// ---- Hardware/NanotecPanDrive/FB_NanotecPD_Home.TcPOU
FUNCTION_BLOCK FB_NanotecPD_Home
VAR_INPUT
	bExecute 	: BOOL;
	bStop		: BOOL;
END_VAR
VAR_OUTPUT
	bBusy 		: BOOL;
	bError 		: BOOL;
	nErrorId 	: ERRORID;	
END_VAR
VAR_IN_OUT
	pHwRef : POINTER TO FB_HwRefNanotecPD; 
END_VAR
VAR
	nState 				: USINT;
	nStateNext			: USINT;
	fbSdoWrite 			: FB_SDO_WRITE;
	eCurrentHomingState : E_CoDS402HomingState;
END_VAR

IF bExecute THEN
	CASE nState OF
		0:	//Set fast homing speed
			bBusy := TRUE;
			fbSdoWrite.nIndex := 16#6099;
			fbSdoWrite.nSubIndex := 1;
			fbSdoWrite.nDataLength := 4;
			fbSdoWrite.nData := pHwRef^.M_RealToInternSpeed(pHwRef^.P_nFastHomingSpeed);
			nState := 40;
			nStateNext := 1;
			
		1:	//Set slow homing speed
			fbSdoWrite.nIndex := 16#6099;
			fbSdoWrite.nSubIndex := 2;
			fbSdoWrite.nDataLength := 4;
			fbSdoWrite.nData := pHwRef^.M_RealToInternSpeed(pHwRef^.P_nSlowHomingSpeed);
			nState := 40;
			nStateNext := 2;
			
		2:	//Set homing methode
			fbSdoWrite.nIndex := 16#6098;
			fbSdoWrite.nSubIndex := 0;
			fbSdoWrite.nDataLength := 1;
			IF pHwRef^.P_bInvertInitDir THEN
				fbSdoWrite.nData := 2;
			ELSE
				fbSdoWrite.nData := 1;
			END_IF
			nState := 40;
			nStateNext := 3;
			
		3: 	//Write home offset
			fbSdoWrite.nIndex := 16#607C;
			fbSdoWrite.nSubIndex := 0;
			fbSdoWrite.nDataLength := 4;
			//Hier braucht es Umrechnung von Real to intern Pos
			fbSdoWrite.nData := pHwRef^.M_RealToInternPos(pHwRef^.P_nRefPos);
			nState := 40;
			IF pHwRef^.M_GetDS402State() = E_CoDS402States.DS402STATE_OperationEnabled THEN
				nStateNext := 4;
			ELSE
				nStateNext := 5;
			END_IF
			
		4:	//Mode lässt sich nicht in "OperationEnabled" setzen
			pHwRef^.nControlword := 7;
			IF pHwRef^.M_GetDS402State() = E_CoDS402States.DS402STATE_SwitchedOn THEN
				nState := 5;	
			END_IF
			
		5:	//Set Mode of operation to "6" (Homing)
			pHwRef^.nMode := 6; //Homing
			IF pHwRef^.nCurrentMode = 6 THEN
				nState := 6;	
			END_IF

		6:	//Statemachine in "OperationEnabled" setzen
			pHwRef^.nControlword := 15;
			IF pHwRef^.M_GetDS402State() = E_CoDS402States.DS402STATE_OperationEnabled THEN
				nState := 7;
			END_IF
			
		7:	//Start homing
			pHwRef^.nControlword := 31;
			eCurrentHomingState := pHwRef^.M_GetHomingState();
			IF eCurrentHomingState = E_CoDS402HomingState.HomingInProgress THEN
				nState := 8;
			END_IF
			
		8:	//Wait for State "Homing in process
			IF pHwRef^.M_GetDS402State() = E_CoDS402States.DS402STATE_OperationEnabled THEN
				IF bStop THEN
					pHwRef^.nControlword := 15;
					nState := 80;
				ELSE
					eCurrentHomingState := pHwRef^.M_GetHomingState();
					CASE eCurrentHomingState OF
						E_CoDS402HomingState.HomingAttainedButNotReached,
						E_CoDS402HomingState.HomingError,
						E_CoDS402HomingState.HomingInteruptedOrNotReached:
							nErrorId := E_ErrorIdDS402.ERRORID_HomingInterruptedOrNotReached;
							nState := 99;
						E_CoDS402HomingState.HomingSuccess:
							pHwRef^.P_bIsHomed := TRUE;
							pHwRef^.nControlword := 7;
							pHwRef^.nMode := 1;
							pHwRef^.nTargetSpeed := DINT_TO_INT(pHwRef^.M_RealToInternSpeed(pHwRef^.P_nFastHomingSpeed));
							pHwRef^.nTargetPosition := pHwRef^.M_RealToInternPos(pHwRef^.P_nHomePos);
							nState := 9;
					END_CASE
				END_IF
			ELSE
				nErrorId := E_ErrorIdDS402.ERRORID_OperationNotEnabled;
				nState := 99;
			END_IF
			
		9:	//Move to WorkingPos1
			IF pHwRef^.nCurrentMode = 1 THEN
				pHwRef^.nControlword := 15;
				nState := 10;
			END_IF
			
		10:	IF pHwRef^.M_GetDS402State() = E_CoDS402States.DS402STATE_OperationEnabled THEN
				pHwRef^.nControlword := 31;
				nState := 11;
			END_IF
			
		11:	//Wait for setpoint acknowledge
			IF pHwRef^.nStatusword.12 THEN
				pHwRef^.nControlword := 15;
				nState := 12;
			END_IF
			
		12:	//Wait for target reached
			IF pHwRef^.M_GetDS402State() = E_CoDS402States.DS402STATE_OperationEnabled THEN
				IF bStop THEN
					pHwRef^.nControlword.8 := TRUE;
					nState := 13;
				ELSE
					IF pHwRef^.nStatusword.10 THEN
						nState := 80;	
					END_IF
				END_IF
			ELSE
				nErrorId := E_ErrorIdDS402.ERRORID_OperationNotEnabled;
				nState := 99;
			END_IF
			
		13:	//Warten bis Motor sich nicht mehr dreht -> dann Power-STM in SwitchedOn setzen, damit Fahrauftrag gelöscht wird
			IF pHwRef^.nCurrentSpeed = 0 THEN
				pHwRef^.nControlword := 7;
				nState := 14;
			END_IF
			
		14:	//Power-STM wieder in OperationEnable setzen
			IF pHwRef^.M_GetDS402State() = E_CoDS402States.DS402STATE_SwitchedOn THEN
				pHwRef^.nControlword := 15;
				pHwRef^.P_bIsHomed := TRUE;
				nState := 80;
			END_IF		

	END_CASE
	
	//Sdo senden
	IF nState = 40 THEN
		fbSdoWrite(sADSNetID:= pHwRef^.P_sAdsNetId, nPortNr:= pHwRef^.P_nAdsPort, bExecute:= TRUE);
		IF NOT fbSdoWrite.bBusy THEN
			IF fbSdoWrite.bError THEN
				nErrorId := fbSdoWrite.nAdsErrorId;
				nState := 99;
			ELSE
				nState := nStateNext;
			END_IF
			fbSdoWrite(bExecute:= FALSE);
		END_IF		
	END_IF
	
	IF nState >= 80 THEN
		bBusy := FALSE;
		IF nState = 99 THEN
			bError := TRUE;
		END_IF
	END_IF
	
ELSE
	bError := FALSE;
	nErrorId := 0;
	nState := 0;	
END_IF

END_FUNCTION_BLOCK

// ---- Hardware/TMCM-1140/FB_TMCM1140_Home.TcPOU
FUNCTION_BLOCK FB_TMCM1140_Home
VAR_INPUT
	bExecute	: BOOL;
	bStop		: BOOL;
END_VAR
VAR_OUTPUT
	bBusy 		: BOOL;
	bError 		: BOOL;
	nErrorId 	: ERRORID;	
END_VAR
VAR_IN_OUT
	pHwRef : POINTER TO FB_HwRefTMCM1140;
END_VAR
VAR
	nState 			: USINT;
	nStateNext 		: USINT;
	bDigiout0 		: BOOL;
	bDigiout1 		: BOOL;
	fbSdoWrite 		: FB_SDO_WRITE;
	eCurrentHomingState : E_CoDS402HomingState;
END_VAR

IF bExecute THEN
	CASE nState OF
		0:	//Set Fast homing speed
			bBusy := TRUE;
			fbSdoWrite.nIndex := 16#6099;
			fbSdoWrite.nSubIndex := 1;
			fbSdoWrite.nDataLength := 4;
			fbSdoWrite.nData := pHwRef^.M_RealToInternSpeed(pHwRef^.P_nFastHomingSpeed);
			nState := 40;
			nStateNext := 1;
			
		1:	//Set Slow homing speed
			fbSdoWrite.nIndex := 16#6099;
			fbSdoWrite.nSubIndex := 2;
			fbSdoWrite.nDataLength := 4;
			fbSdoWrite.nData := pHwRef^.M_RealToInternSpeed(pHwRef^.P_nSlowHomingSpeed);
			nState := 40;
			nStateNext := 2;			

		2:	//Set homing methode
			fbSdoWrite.nIndex := 16#6098;
			fbSdoWrite.nSubIndex := 0;
			fbSdoWrite.nDataLength := 1;
			fbSdoWrite.nData := pHwRef^.P_eHomingMethode;
			nState := 40;
			nStateNext := 3;
			
		3: 	//Write home offset
			fbSdoWrite.nIndex := 16#607C;
			fbSdoWrite.nSubIndex := 0;
			fbSdoWrite.nDataLength := 4;
			fbSdoWrite.nData := pHwRef^.M_RealToInternPos(pHwRef^.P_nRefPos);
			nState := 40;
			nStateNext := 4;
			
		4:	//Write profile speed
			fbSdoWrite.nIndex := 16#6081;
			fbSdoWrite.nSubIndex := 0;
			fbSdoWrite.nDataLength := 4;
			fbSdoWrite.nData := pHwRef^.M_RealToInternSpeed(pHwRef^.P_nMaxSpeed);
			nState := 40;
			nStateNext := 5;

		5:	//Set Mode of operation to "6" (Homing)
			pHwRef^.nMode := 6; //Homing
			nState := 6;
			
		6:	//Start homing
			pHwRef^.nControlword := 31;
			nState := 7;
			
		7:	//Wait for State "Homing in process
			IF pHwRef^.M_GetDS402State() = E_CoDS402States.DS402STATE_OperationEnabled THEN
				IF bStop THEN
					pHwRef^.nControlword := 15;
					nState := 80;
				ELSE
					eCurrentHomingState := pHwRef^.M_GetHomingState();
					CASE eCurrentHomingState OF
						E_CoDS402HomingState.HomingAttainedButNotReached,
						E_CoDS402HomingState.HomingError,
						E_CoDS402HomingState.HomingInteruptedOrNotReached:
							nErrorId := E_ErrorIdDS402.ERRORID_HomingInterruptedOrNotReached;
							nState := 99;
						E_CoDS402HomingState.HomingSuccess:
							pHwRef^.nControlword := 15;
							pHwRef^.nMode := 1;	//PP mode
							pHwRef^.M_SetTargetPos(pHwRef^.P_nHomePos, FALSE);
							pHwRef^.P_bIsHomed := TRUE;
							nState := 8;
					END_CASE
				END_IF
			ELSE
				nErrorId := 43434;
				nState := 99;
			END_IF
			
		8:	//Move to HomePos
			pHwRef^.nControlword := 31;
			nState := 9;
			
		9:	//Wait for setpoint acknowledge
			IF pHwRef^.nStatusword.12 THEN
				pHwRef^.nControlword := 15;
				nState := 10;
			END_IF
			
		10:	//Wait for target reached
			IF pHwRef^.M_GetDS402State() = E_CoDS402States.DS402STATE_OperationEnabled THEN
				//Das HALT-Bit von von der TMCM1140 nicht unterstützt.
				//Man kann den Mode auf "0" setzen und dann sollter der Motor auch anhalten
				IF bStop THEN
					IF bStop THEN
						pHwRef^.nMode := 0;
						nState := 80;
					END_IF
				ELSE
					IF pHwRef^.nStatusword.10 THEN
						nState := 80;
					END_IF
				END_IF
			ELSE
				nErrorId := E_ErrorIdDS402.ERRORID_OperationNotEnabled;
				nState := 99;
			END_IF
			
	END_CASE
	
	//Sdo senden
	IF nState = 40 THEN
		fbSdoWrite(sADSNetID:= pHwRef^.P_sAdsNetId, nPortNr:= pHwRef^.P_nAdsPort, bExecute:= TRUE);
		IF NOT fbSdoWrite.bBusy THEN
			IF fbSdoWrite.bError THEN
				nErrorId := fbSdoWrite.nAdsErrorId;
				nState := 99;
			ELSE
				nState := nStateNext;
			END_IF
			fbSdoWrite(bExecute:= FALSE);
		END_IF		
	END_IF
	
	IF nState >= 80 THEN
		bBusy := FALSE;
		IF nState = 99 THEN
			bError := TRUE;
		END_IF
	END_IF

ELSE
	bBusy 	:= FALSE;
	bError 	:= FALSE;
	bStop 	:= FALSE;
	nState 	:= 0;
END_IF

END_FUNCTION_BLOCK

// ---- Hardware/NanotecPanDrive/FB_NanotecPD_Move.TcPOU
FUNCTION_BLOCK FB_NanotecPD_Move
VAR_INPUT
	bExecute 	: BOOL;
	bStop		: BOOL;
	nPosition	: DINT; //Reale Einheit (µm oder 1/10°)
	nSpeed		: DINT; //Reale Einheit/s	
END_VAR
VAR_OUTPUT
	bBusy 		: BOOL;
	bError 		: BOOL;
	nErrorId 	: ERRORID;	
END_VAR
VAR_IN_OUT
	pHwRef : POINTER TO FB_HwRefNanotecPD; 
END_VAR
VAR
	nState 					: USINT;
	eCurrentCoDS402State 	: E_CoDS402States;
	fbGetCurrTaskIndex		: GETCURTASKINDEX;
	nCurrentTaskCycleCount 	: UDINT;	
END_VAR

IF bExecute THEN
	eCurrentCoDS402State := pHwRef^.M_GetDS402State();
	
	CASE nState OF
		0:	//Vorbedingungen prüfen
			bBusy := TRUE;
			nState := 1;
			IF pHwRef^.bError THEN
				nErrorID := E_ErrorIdHwGeneral.ERRORID_DriveIsInErrorState;
				nState := 99;
			ELSE
				IF pHwRef^.bBusy THEN
					nErrorID := E_ErrorIdHwGeneral.ERRORID_DriveIsStillBusy;
					nState := 99;
				ELSE
					IF NOT pHwRef^.P_bIsHomed THEN
						nErrorID := E_ErrorIdHwGeneral.ERRORID_DriveNotHomed;
						nState := 99;
					ELSE
						IF NOT pHwRef^.M_SetTargetPos(nPosition) THEN
							nErrorID := E_ErrorIdHwGeneral.ERRORID_InvalidPosition;
							nState := 99;
						ELSE
							IF NOT pHwRef^.M_SetTargetSpeed(nSpeed) THEN
								nErrorID := E_ErrorIdHwGeneral.ERRORID_InvalidSpeed;
								nState := 99;
							END_IF
						END_IF	
					END_IF
				END_IF
			END_IF
			
			fbGetCurrTaskIndex();
			nCurrentTaskCycleCount := TwinCAT_SystemInfoVarList._TaskInfo[fbGetCurrTaskIndex.index].CycleCount;

		1:	//Mode sollte durch Homing bereits auf 1 stehen
			//Dieser State darf niemals im gleichen Zyklus wie State 0 ausgeführt werden. Passiert wenn FB im selben Zyklus auf-
			//gerufen wird. Somit wird sichergestellt, dass die Zielposition auch im Drive eher ankommt, wie das Startbit.
			IF TwinCAT_SystemInfoVarList._TaskInfo[fbGetCurrTaskIndex.index].CycleCount <> nCurrentTaskCycleCount THEN
				IF eCurrentCoDS402State = E_CoDS402States.DS402STATE_OperationEnabled THEN
					pHwRef^.nControlword := 31;
					nState := 2;
				ELSE
					nErrorID := E_ErrorIdDS402.ERRORID_OperationNotEnabled;
					nState := 99;
				END_IF
			END_IF
			
		2:	//Setpoint ACK?
			IF pHwRef^.nStatusword.12 THEN
				pHwRef^.nControlword := 15;
				nState := 3;
			END_IF
			
		3:	//Target reached?
			IF pHwRef^.bError THEN
				nErrorId := pHwRef^.P_nErrorID;
				nState := 99;
			ELSE
				{warning 'Safety sollte noch mit abgefragt werden'}
				IF bStop THEN
					pHwRef^.nControlword.8 := TRUE;
					nState := 4;
				END_IF
				
				IF pHwRef^.nStatusword.10 THEN
					nState := 80; //Ready
				END_IF
			END_IF
			
		4:	//Warten bis Motor sich nicht mehr dreht -> dann OperationEnable zurück nehmen
			IF pHwRef^.nCurrentSpeed = 0 THEN
				pHwRef^.nControlword := 7;
				nState := 5;
			END_IF			
			
		5:	//STM wieder in OperationEnable
			IF pHwRef^.M_GetDS402State() = E_CoDS402States.DS402STATE_SwitchedOn THEN
				pHwRef^.nControlword := 15;
				nState := 80; //Ready
			END_IF
	END_CASE
	
	IF nState >= 80 THEN
		bBusy := FALSE;
		IF nState = 99 THEN
			bError := TRUE;
		END_IF
	END_IF
	
ELSE
	bError := FALSE;
	nErrorId := 0;
	nState := 0;
END_IF

END_FUNCTION_BLOCK

// ---- Hardware/TrayLock/FB_HwTrayLockControl.TcPOU
FUNCTION_BLOCK FB_HwTrayLockControl
VAR_INPUT
	bExecute		: BOOL;
	eCtrl			: E_LockCtrl;
END_VAR
VAR_OUTPUT
	bBusy 		: BOOL;
	bError 		: BOOL;
	nErrorId	: ERRORID;	
END_VAR
VAR_IN_OUT
	pHwRef : POINTER TO FB_HwRefTrayLock;
END_VAR
VAR
	nState		: USINT;
	timer		: TON;
END_VAR

IF bExecute THEN
	IF pHwRef = 0 THEN
		bError := TRUE;
		nErrorId := E_ErrorIdHwGeneral.ERRORID_InvalidHwRef;
		RETURN;
	END_IF

	CASE nState OF
		0:	IF eCtrl = E_LockCtrl.Unlock THEN
				IF pHwRef^.eCurrentState = E_LockState.Unlocked THEN
					RETURN;
				ELSE
					bBusy := TRUE;
					nState := 1; //Unlocking
				END_IF
			ELSE
				IF pHwRef^.eCurrentState = E_LockState.Locked THEN
					RETURN;
				ELSE
					bBusy := TRUE;
					nState := 10; //Locking
				END_IF
			END_IF
			
		1:	//Unlocking, disable heater
			pHwRef^.bDisableHeater := TRUE;
			timer(IN:= TRUE, PT:= T#200MS);
			nState := 2;
			
		2:	//Time elapsed?
			timer();
			IF timer.Q THEN
				timer(IN:= FALSE);
				nState := 3;
			END_IF
			
		3:	//Set outputs
			pHwRef^.bLock := FALSE;
			pHwRef^.bUnlock := TRUE;
			timer(IN:= TRUE, PT:= T#3S); //Timeout
			IF pHwRef^.P_bFeedback THEN
				IF pHwRef^.bUnlocked THEN
					nState := 80;
				ELSIF timer.Q THEN
					nErrorId := E_ErrorIdHwGeneral.ERRORID_UnlockingFailed;
					nState := 99; //Error
				END_IF
			ELSE
				IF timer.Q THEN
					nState := 80;
				END_IF
			END_IF
			
		10: //Locking
			pHwRef^.bLock := TRUE;
			pHwRef^.bUnlock := FALSE;
			timer(IN:= TRUE, PT:= T#3S); //Timeout
			IF pHwRef^.P_bFeedback THEN
				IF pHwRef^.bLocked THEN
					//Enable heater
					pHwRef^.bDisableHeater := FALSE;
					nState := 80;
				ELSIF timer.Q THEN
					nErrorId := E_ErrorIdHwGeneral.ERRORID_LockingFailed;
					nState := 99; //Error
				END_IF
			ELSE
				IF timer.Q THEN
					nState := 80;
				END_IF
			END_IF
	END_CASE
	
	IF nState >= 80 THEN
		pHwRef^.bLock := FALSE;
		pHwRef^.bUnlock := FALSE;
		bBusy := FALSE;
		IF nState = 99 THEN
			bError := TRUE;
		END_IF
	END_IF

ELSE
	timer(IN:= FALSE);
	bBusy := FALSE;
	bError := FALSE;
	nErrorId := 0;
	nState := 0;	
END_IF

END_FUNCTION_BLOCK

// ---- Objects/Devices/FB_Stacker.TcPOU
FUNCTION_BLOCK FB_Stacker EXTENDS FB_Object IMPLEMENTS I_Device

VAR
	nParentSlotNr		: UINT;		//Stacker befindet sich zwar an keinem Slot, aber virtuell in der GUI (am Root)#
	eCurrentState		: E_MachineState := E_MachineState.MACHINESTATE_Idle;
	nNotifyId			: UINT;
	nErrorId			: ERRORID;
	bCanceled			: BOOL;
	bStopAllOnError		: BOOL;
	bIsInit				: BOOL;
	bBusy				: BOOL;
	bError				: BOOL;
	stError				: ST_Error :=(POU := E_POU.POU_FB_Stacker);
	
	nNumberOfShelves	: USINT;
	aShelfes			: ARRAY[1..cMaxShelfes] OF ST_Shelf;
	
	//Hardware-Referenzen
	pHwRef_SpinDrive	: POINTER TO FB_HwRefEL70xxDrive;
	pHwRef_LiftDrive	: POINTER TO FB_HwRefEL70xxDrive;
	pHwRef_TrayStop		: POINTER TO FB_HwRefEL70xxDrive;
	
	bSensorTransAreaLeft 		AT %I* : BOOL;
	bSensorTransAreaRight		AT %I* : BOOL;
	bSensorTrayAlignmentLeft 	AT %I* : BOOL;
	bSensorTrayAlignmentRight 	AT %I* : BOOL;
	bSensorTrayDetection		AT %I* : BOOL;
	
	//Spec-Properties
	nLoadingPosAngle		: DINT;	//Drehwinkel Beladeposition
	nTransferPosAnglePrint1 : DINT;	//Drehwinkel Transferpostion zu Drucker 1
	nTransferPosAnglePrint2 : DINT;	//Drehwinkel Transferpostion zu Drucker 2 (wird derzeit nicht verwendet)
		
	//****************************************Aktionvariablen****************************************************
	
	//Action: "Init"
	bInit				: BOOL;
	nStateA_Init		: USINT;
	fbPower 			: FB_HWECtrl_EL70xx_Power;
	fbHoming 			: FB_HWECtrl_EL70xx_Home;
	pCurrentInitDrive	: POINTER TO FB_HwRefEL70xxDrive;
	
	//Action: "TurnTo"
	bTurnTo				: BOOL;
	nStateA_TurnTo		: USINT;
	fbHwCtrl_Turn		: FB_HWECtrl_EL70xx_Move;
	nTurnToPosition		: DINT;
	
	//Action: "MoveLifter"
	bMoveLifter			: BOOL;
	nStateA_MoveLifter	: USINT;
	nMoveLifterPosition	: DINT;
	nMoveLifterSpeed	: DINT;
	fbHWECtrl_MoveLifter: FB_HWECtrl_EL70xx_Move;
	
	//Action: "OpenCloseTrayStop"
	bOpClTrayStop			: BOOL;
	nStateA_OpClTrayStop	: USINT;
	eOpClTrayStopCtrl		: E_OpClCtrl;
	fbHwCtrl_MoveTrayStop 	: FB_HWECtrl_EL70xx_Move;
	
	//Action: "Load" (Bestücken oder Entnehmen)
	bLoad			: BOOL;
	nStateA_Load	: USINT;
	nBottomShelf	: UINT; //unterstes Fach
	
	stProcessData		: ST_ObjectProcData;
	
END_VAR

VAR CONSTANT
	cMaxShelfes : UINT := 10;
END_VAR

CASE eCurrentState OF
	E_MachineState.MACHINESTATE_Active:
	
		IF bInit THEN
			A_Init();
			IF nStateA_Init >= 80 THEN
				IF nStateA_Init >= 99 THEN
					bError := TRUE;	
				END_IF
				bInit := FALSE;
				nStateA_Init := 0;
			END_IF
		END_IF
		
		IF bTurnTo THEN
			A_TurnTo();
			IF nStateA_TurnTo >= 80 THEN
				IF nStateA_TurnTo >= 99 THEN
					bError := TRUE;	
				END_IF
				bTurnTo := FALSE;
				nStateA_TurnTo := 0;
			END_IF
		END_IF
		
		IF bMoveLifter THEN
			A_MoveLifter();
			IF nStateA_MoveLifter >= 80 THEN
				IF nStateA_MoveLifter >= 99 THEN
					bError := TRUE;	
				END_IF
				bMoveLifter := FALSE;
				nStateA_MoveLifter := 0;
			END_IF
		END_IF
		
		IF bOpClTrayStop THEN
			A_OpClTrayStop();
			IF nStateA_OpClTrayStop >= 80 THEN
				IF nStateA_OpClTrayStop >= 99 THEN
					bError := TRUE;	
				END_IF
				bOpClTrayStop := FALSE;
				nStateA_OpClTrayStop := 0;
			END_IF
		END_IF
		
		IF bLoad THEN
			A_Load();
			IF nStateA_Load >= 80 THEN
				IF nStateA_Load >= 99 THEN
					bError := TRUE;	
				END_IF
				bLoad := FALSE;
				nStateA_Load := 0;
			END_IF
		END_IF
		
		IF NOT (bInit OR bTurnTo OR bMoveLifter OR bOpClTrayStop OR bLoad) THEN
			bBusy := FALSE;
			eCurrentState := E_MachineState.MACHINESTATE_Idle;
		END_IF

		IF bError  THEN
			eCurrentState := E_MachineState.MACHINESTATE_Error;
		END_IF

	E_MachineState.MACHINESTATE_Reset:
		nStateA_Init := 0;
		nStateA_TurnTo := 0;
		nStateA_MoveLifter := 0;
		nStateA_OpClTrayStop := 0;
		nStateA_Load := 0;
		bBusy := FALSE;
		bError := FALSE;
		bStopAllOnError := FALSE;
		stError.Cmd := 0;
		stError.ErrorId := 0;
		eCurrentState := E_MachineState.MACHINESTATE_Idle;
	
	E_MachineState.MACHINESTATE_Error:
		bBusy := FALSE;
END_CASE

//Prozessdaten aktualisieren
stProcessData.nObjId := nObjectID;
stProcessData.n32Data[0] := BOOL_TO_DINT(P_bIsInit);
stProcessData.n32Data[1] := eCurrentState;
stProcessData.n32Data[2] := stError.ErrorId;
stProcessData.n32Data[3] := pHwRef_LiftDrive^.P_nActualPosition;
stProcessData.n32Data[4] := pHwRef_SpinDrive^.P_nActualPosition;
IF pHwRef_TrayStop^.bInput1 THEN //Open
	stProcessData.n32Data[5] := E_OpClState.Open;
ELSIF pHwRef_TrayStop^.bInput2 THEN //Closed
	stProcessData.n32Data[5] := E_OpClState.Closed;
ELSE
	stProcessData.n32Data[5] := E_OpClState.UNDEFINED;
END_IF
	stProcessData.n32Data[6] := BOOL_TO_DINT(bSensorTrayAlignmentLeft AND bSensorTrayAlignmentRight);

aObjProcData[nNotifyId] := stProcessData;

ACTION A_Init:
stError.POUState := nStateA_Init;

CASE nStateA_Init OF
	0:	//Power TrayStop
		pCurrentInitDrive := pHwRef_TrayStop;
		fbPower(pHwRef:= pHwRef_TrayStop, bEnable:= TRUE, bExecute:= TRUE);
		IF NOT fbPower.bBusy THEN
			IF fbPower.bError THEN
				stError.ErrorId := fbPower.nErrorId;
				nStateA_Init := 99;
			ELSE
				nStateA_Init := 1;
			END_IF
			fbPower(pHwRef := pHwRef_TrayStop, bExecute:= FALSE);
		END_IF
		
	1:	//Power SpinDrive
		pCurrentInitDrive := pHwRef_SpinDrive;
		fbPower(pHwRef:= pHwRef_SpinDrive, bEnable:= TRUE, bExecute:= TRUE);
		IF NOT fbPower.bBusy THEN
			IF fbPower.bError THEN
				stError.ErrorId := fbPower.nErrorId;
				nStateA_Init := 99;
			ELSE
				nStateA_Init := 2;
			END_IF
			fbPower(pHwRef:= pHwRef_SpinDrive, bExecute:= FALSE);
		END_IF

	2:	//Power LiftDrive
		pCurrentInitDrive := pHwRef_LiftDrive;
		fbPower(pHwRef:= pHwRef_LiftDrive, bEnable:= TRUE, bExecute:= TRUE);
		IF NOT fbPower.bBusy THEN
			IF fbPower.bError THEN
				stError.ErrorId := fbPower.nErrorId;
				nStateA_Init := 99;
			ELSE
				nStateA_Init := 3;
			END_IF
			fbPower(pHwRef:= pHwRef_LiftDrive, bExecute:= FALSE);
		END_IF
		
	3:	//Homing TrayStop
		pCurrentInitDrive := pHwRef_TrayStop;
		fbHoming(pHwRef:= pHwRef_TrayStop, bExecute:= TRUE);
		IF NOT fbHoming.bBusy THEN
			IF fbHoming.bError THEN
				stError.ErrorId := fbHoming.nErrorId;
				nStateA_Init := 99;
			ELSE
				nStateA_Init := 4;
			END_IF
			fbHoming(pHwRef:= pHwRef_TrayStop, bExecute:= FALSE);
		END_IF

	4:	//Homing SpinDrive
		pCurrentInitDrive := pHwRef_SpinDrive;
		fbHoming(pHwRef:= pHwRef_SpinDrive, bExecute:= TRUE);
		IF NOT fbHoming.bBusy THEN
			IF fbHoming.bError THEN
				stError.ErrorId := fbHoming.nErrorId;
				nStateA_Init := 99;
			ELSE
				nStateA_Init := 5;
			END_IF
			fbHoming(pHwRef:= pHwRef_SpinDrive, bExecute:= FALSE);
		END_IF
		
	5:	//Homing LiftDrive
		pCurrentInitDrive := pHwRef_LiftDrive;
		//TransArea überwachen
		IF NOT P_bTransAreaFree THEN
			//Stoppen und dann in Error
			fbHoming(pHwRef:= pHwRef_LiftDrive, bStop := TRUE);
			nStateA_Init := 75;
		ELSE
			fbHoming(pHwRef:= pHwRef_LiftDrive, bExecute:= TRUE);
			IF NOT fbHoming.bBusy THEN
				IF fbHoming.bError THEN
					stError.ErrorId := fbHoming.nErrorId;
					nStateA_Init := 99;
				ELSE
					nStateA_Init := 80;
				END_IF
				fbHoming(pHwRef:= pHwRef_LiftDrive, bExecute:= FALSE);
			END_IF
		END_IF
		
	70:	//Abbrechen
		IF fbPower.bBusy THEN //Warten bis fbPower fertig
			nStateA_Init := 71;
		ELSIF fbHoming.bBusy THEN
			nStateA_Init := 72;
		ELSE
			nStateA_Init := 80;
		END_IF
		
	71:	//Power ready?
		fbPower(pHwRef:= pCurrentInitDrive);
		IF NOT fbPower.bBusy THEN
			fbPower(pHwRef:= pCurrentInitDrive, bExecute := FALSE);
			nStateA_Init := 80;
		END_IF
		
	72:	//Homing abbrechen
		fbHoming(pHwRef:= pCurrentInitDrive, bStop:= TRUE);
		IF NOT fbHoming.bBusy THEN
			fbHoming(pHwRef:= pCurrentInitDrive, bStop:= FALSE, bExecute := FALSE);
			nStateA_Init := 80;
		END_IF
		
	75:	//Homing Lifter abbrechen und dann in Error
		fbHoming(pHwRef:= pCurrentInitDrive, bStop:= TRUE);
		IF NOT fbHoming.bBusy THEN
			fbHoming(pHwRef:= pCurrentInitDrive, bStop:= FALSE, bExecute := FALSE);
			stError.ErrorId := E_ErrorIdCmd.ERRORID_TransferAreaNotFree;
			nStateA_Init := 99;
		END_IF
 	
END_CASE

//Errorhandling
IF nStateA_Init = 99 THEN
	stError.ObjectId := nObjectID;
	stError.Cmd := E_Action.ACTION_Init;
	stError.POUAction := E_POUACT.POUACT_A_Init;
	fbErrorList.M_Add(stError);
END_IF
END_ACTION

ACTION A_Load:
//Diese Action darf nur ausgeführt werden, wenn:
//Initialisiert ist
//keine andere Action aktiv ist
//Es werden alle Actions einzeln ausgeführt.
//1. turn
//2. move lifter
//3. close tray stopper
//4. open interlock

CASE nStateA_Load OF
	0:	//Turn to loading position
		nTurnToPosition := nLoadingPosAngle;
		A_TurnTo();
		IF nStateA_TurnTo >= 80 THEN
			IF nStateA_TurnTo >= 99 THEN
				nStateA_Load := 99;
			ELSE
				nStateA_Load := 1;
			END_IF
			nStateA_TurnTo := 0;
		END_IF

	1:	//Move lifter
		nMoveLifterPosition := M_GetBottomShelfPos();
		nMoveLifterSpeed := pHwRef_LiftDrive^.P_nMaxSpeed;
		A_MoveLifter();
		IF nStateA_MoveLifter >= 80 THEN
			IF nStateA_MoveLifter >= 99 THEN
				nStateA_Load := 99;
			ELSE
				nStateA_Load := 2;
			END_IF
			nStateA_MoveLifter := 0;
		END_IF
				
	2:	//Close tray stopper
		eOpClTrayStopCtrl := E_OpClCtrl.Close;
		A_OpClTrayStop();
		IF nStateA_OpClTrayStop >= 80 THEN
			IF nStateA_OpClTrayStop >= 99 THEN
				nStateA_Load := 99;
			ELSE
				nStateA_Load := 3;
			END_IF
			nStateA_OpClTrayStop := 0;
		END_IF
		
	3:	//Open interlock stacker
		{IF defined(Stacker)}
		fbSafetyStacker.M_Control(E_SafetyCtrl.Unlock);
		{END_IF}
		nStateA_Load := 80;
	
	70:	//Cancel
		//Which actin is active?
		//we can identify the active action wich nStateA_xxxx is greather than 0
		IF nStateA_TurnTo > 0 THEN
			;
		ELSIF nStateA_MoveLifter > 0 THEN
			;
		ELSIF nStateA_OpClTrayStop > 0 THEN
			;
		END_IF
	
	
END_CASE
END_ACTION

ACTION A_MoveLifter:
IF nStateA_MoveLifter = 0 THEN
	//Nur TransArea überwachen	
	IF NOT P_bTransAreaFree THEN
		//Stoppen und dann in Error
		fbHWECtrl_MoveLifter(pHwRef:= pHwRef_LiftDrive, bStop:= TRUE);
		nStateA_MoveLifter := 75;
	ELSE
		fbHWECtrl_MoveLifter(pHwRef:= pHwRef_LiftDrive, nPosition := nMoveLifterPosition, nSpeed:= nMoveLifterSpeed, bExecute:= TRUE);
		IF NOT fbHWECtrl_MoveLifter.bBusy THEN
			IF fbHWECtrl_MoveLifter.bError THEN
				stError.ErrorId := fbHWECtrl_MoveLifter.nErrorId;
				nStateA_MoveLifter := 99;
			ELSE
				nStateA_MoveLifter := 80;
			END_IF
			fbHWECtrl_MoveLifter(pHwRef:= pHwRef_LiftDrive, bExecute:= FALSE);
		END_IF
	END_IF
	
ELSIF nStateA_MoveLifter = 70 THEN //Normal stoppen
	fbHWECtrl_MoveLifter(pHwRef:= pHwRef_LiftDrive, bStop := TRUE);
	IF NOT fbHWECtrl_MoveLifter.bBusy THEN
		IF fbHWECtrl_MoveLifter.bError THEN
			stError.ErrorId := fbHWECtrl_MoveLifter.nErrorId;
			nStateA_MoveLifter := 99;
		ELSE
			nStateA_MoveLifter := 80;
		END_IF
		fbHWECtrl_MoveLifter(pHwRef:= pHwRef_LiftDrive, bExecute:= FALSE);
	END_IF
	
ELSIF nStateA_MoveLifter = 75 THEN //Stoppen mit folgender Error-Meldung
	fbHWECtrl_MoveLifter(pHwRef:= pHwRef_LiftDrive);
	IF NOT fbHWECtrl_MoveLifter.bBusy THEN
		IF fbHWECtrl_MoveLifter.bError THEN
			stError.ErrorId := fbHWECtrl_MoveLifter.nErrorId;
		ELSE
			stError.ErrorId := E_ErrorIdCmd.ERRORID_TransferAreaNotFree;
		END_IF
		fbHWECtrl_MoveLifter(pHwRef:= pHwRef_LiftDrive, bExecute:= FALSE);
		nStateA_MoveLifter := 99;
	END_IF
END_IF

//Errorhandling
IF nStateA_MoveLifter = 99 THEN
	stError.ObjectId := nObjectID;
	stError.Cmd := E_Action.ACTION_MoveLifter;
	stError.POUAction := E_POUACT.POUACT_A_MoveLifter;
	fbErrorList.M_Add(stError);
END_IF
END_ACTION

ACTION A_OpClTrayStop:
IF nStateA_OpClTrayStop = 0 THEN
	IF eOpClTrayStopCtrl = E_OpClCtrl.Close THEN
		fbHwCtrl_MoveTrayStop(pHwRef:= pHwRef_TrayStop, nPosition:= pHwRef_TrayStop^.P_nMaxPos, nSpeed:= pHwRef_TrayStop^.P_nMaxSpeed, bExecute:= TRUE);
		nStateA_OpClTrayStop := 1;
	ELSE
		fbHwCtrl_MoveTrayStop(pHwRef:= pHwRef_TrayStop, nPosition:= 0, nSpeed:= pHwRef_TrayStop^.P_nMaxSpeed, bExecute:= TRUE);
		nStateA_OpClTrayStop := 1;
	END_IF
ELSIF nStateA_OpClTrayStop = 1 THEN
	fbHwCtrl_MoveTrayStop(pHwRef:= pHwRef_TrayStop);
	IF NOT fbHwCtrl_MoveTrayStop.bBusy THEN
		IF fbHwCtrl_MoveTrayStop.bError THEN
			stError.ErrorId := fbHwCtrl_MoveTrayStop.nErrorId;
			nStateA_OpClTrayStop := 99;
		ELSE
			IF eOpClTrayStopCtrl = E_OpClCtrl.Close THEN
				IF pHwRef_TrayStop^.bInput2 THEN
					nStateA_OpClTrayStop := 80;
				ELSE
					stError.ErrorId := E_ErrorIdCmd.ERRORID_TrayStopNotClosed;
					nStateA_OpClTrayStop := 99;
				END_IF
			ELSE
				IF pHwRef_TrayStop^.bInput1 THEN
					nStateA_OpClTrayStop := 80;
				ELSE
					stError.ErrorId := E_ErrorIdCmd.ERRORID_TrayStopNotOpen;
					nStateA_OpClTrayStop := 99;
				END_IF
			END_IF
		END_IF
		fbHwCtrl_MoveTrayStop(pHwRef:= pHwRef_TrayStop, bExecute:= FALSE);
	END_IF
ELSIF nStateA_OpClTrayStop = 70 THEN
	fbHwCtrl_MoveTrayStop(pHwRef:= pHwRef_TrayStop, bStop := TRUE);
	IF NOT fbHwCtrl_MoveTrayStop.bBusy THEN
		IF fbHwCtrl_MoveTrayStop.bError THEN
			stError.ErrorId := fbHwCtrl_MoveTrayStop.nErrorId;
			nStateA_OpClTrayStop := 99;
		ELSE
			nStateA_OpClTrayStop := 80;
		END_IF
		fbHwCtrl_MoveTrayStop(pHwRef:= pHwRef_TrayStop, bExecute:= FALSE);
	END_IF
	
END_IF

//Errorhandling
IF nStateA_OpClTrayStop = 99 THEN
	stError.ObjectId := nObjectID;
	stError.Cmd := E_Action.ACTION_OpenClose;
	stError.POUAction := E_POUACT.POUACT_A_OpClTrayStop;
	fbErrorList.M_Add(stError);
END_IF
END_ACTION

ACTION A_TurnTo:
IF nStateA_TurnTo = 0 THEN
	fbHwCtrl_Turn(pHwRef:= pHwRef_SpinDrive, nPosition:= nTurnToPosition, nSpeed:= pHwRef_SpinDrive^.P_nMaxSpeed,
					nToleranceWindow:= 50, bExecute:= TRUE);
	IF NOT fbHwCtrl_Turn.bBusy THEN
		IF fbHwCtrl_Turn.bError THEN
			stError.ErrorId := fbHwCtrl_Turn.nErrorId;
			nStateA_TurnTo := 99;
		ELSE
			nStateA_TurnTo := 80;
		END_IF
		fbHwCtrl_Turn(pHwRef:= pHwRef_SpinDrive, bExecute := FALSE);
	END_IF
ELSIF nStateA_TurnTo = 70 THEN
	fbHwCtrl_Turn(pHwRef:= pHwRef_SpinDrive, bStop:= TRUE);
	IF NOT fbHwCtrl_Turn.bBusy THEN
		IF fbHwCtrl_Turn.bError THEN
			stError.ErrorId := fbHwCtrl_Turn.nErrorId;
			nStateA_TurnTo := 99;
		ELSE
			nStateA_TurnTo := 80;
		END_IF
		fbHwCtrl_Turn(pHwRef:= pHwRef_SpinDrive, bExecute := FALSE);
	END_IF	
END_IF

//Errorhandling
IF nStateA_TurnTo = 99 THEN
	stError.ObjectId := nObjectID;
	stError.Cmd := E_Action.ACTION_TurnTo;
	stError.POUAction := E_POUACT.POUACT_A_TurnTo;
	fbErrorList.M_Add(stError);
END_IF
END_ACTION

METHOD FB_init : BOOL
VAR_INPUT
	bInitRetains 		: BOOL; // if TRUE, the retain variables are initialized (warm start / cold start)
	bInCopyCode 		: BOOL;  // if TRUE, the instance afterwards gets moved into the copy code (online change)
END_VAR
eObjectType := E_ObjectType.OBJECTTYPE_Stacker;
eObjectGroup := E_ObjectGroup.OBJECTGROUP_Device;
END_METHOD

METHOD M_CancelAction
VAR_INPUT
	eAction : E_Action;
END_VAR
CASE eAction OF
	E_Action.ACTION_Init:
		IF bInit AND nStateA_Init < 70 THEN
			nStateA_Init := 70;
		END_IF
		
	E_Action.ACTION_TurnTo:
		IF bTurnTo AND nStateA_TurnTo < 70 THEN
			nStateA_TurnTo := 70;
		END_IF
		
	E_Action.ACTION_MoveLifter:
		IF bMoveLifter AND nStateA_MoveLifter < 70 THEN
			nStateA_MoveLifter := 70;
		END_IF
		
	E_Action.ACTION_OpenClose:
		IF bOpClTrayStop AND nStateA_OpClTrayStop < 70 THEN
			nStateA_OpClTrayStop := 70;
		END_IF
		
END_CASE
END_METHOD

METHOD M_CheckAction : ERRORID
VAR_INPUT
	refActionData 	: REFERENCE TO ST_ActionData;
	pCorrelObject	: POINTER TO FB_Object;
END_VAR
M_CheckAction := E_ErrorIdCmd.ERRORID_InvalidAction;
END_METHOD

METHOD M_CheckProcDataType : BOOL
VAR_INPUT
	eProcDataType : E_ProcDataType;
END_VAR
END_METHOD

METHOD M_ClearAllProps
VAR_INPUT
	bIgnoreParent : BOOL; //Es wird das gesamte OD gelöscht. -> Zeiger auf Parent nicht mehr gültig!	
END_VAR
MEMSET(ADR(aShelfes), 0, SIZEOF(aShelfes));
END_METHOD

METHOD M_ExeAction : ERRORID
VAR_INPUT
	refActionData	: REFERENCE TO ST_ActionData;
END_VAR


VAR
	eStackerRotPosition : E_StackerRotPosition;
END_VAR
//Stacker ist so implementiet, dass mehrere Actions nicht zeitgleich ausgeführt werden können.
//Das bedeutet, dass eCurrentState idle sein muss
IF eCurrentState = E_MachineState.MACHINESTATE_Active THEN
	M_ExeAction := E_ErrorIdCmd.ERRORID_BasicActionActive;
	RETURN;	
ELSIF eCurrentState = E_MachineState.MACHINESTATE_Error OR eCurrentState = E_MachineState.MACHINESTATE_Reset THEN
	M_ExeAction := E_ErrorIdCmd.ERRORID_InvalidState;
	RETURN;	
END_IF

IF refActionData.eAction <> E_Action.ACTION_Init THEN
	IF NOT P_bIsInit THEN
		M_ExeAction := E_ErrorIdCmd.ERRORID_DeviceNotInitialized;
		RETURN;
	END_IF
END_IF

{IF defined(Stacker)}
IF fbSafetyStacker.eCurrentState <> E_SafetyState.Locked THEN
	M_ExeAction := E_ErrorIdCmd.ERRORID_InterlockNotLocked;
END_IF
{END_IF}

CASE refActionData.eAction OF
	E_Action.ACTION_Init:
		IF NOT bInit THEN
			IF NOT P_bTransAreaFree THEN
				M_ExeAction := E_ErrorIdCmd.ERRORID_TransferAreaNotFree;
				RETURN;
			END_IF
			
			IF NOT P_bTraysAligned THEN
				M_ExeAction := E_ErrorIdCmd.ERRORID_TraysNotAligned;
				RETURN;
			END_IF
			bInit := TRUE;
		ELSE
			RETURN;
		END_IF

	E_Action.ACTION_TurnTo:
		IF NOT bTurnTo THEN
			IF NOT P_bTransAreaFree THEN
				M_ExeAction := E_ErrorIdCmd.ERRORID_TransferAreaNotFree;
				RETURN;
			END_IF
			
			IF NOT P_bTraysAligned THEN
				M_ExeAction := E_ErrorIdCmd.ERRORID_TraysNotAligned;
				RETURN;
			END_IF
			
			eStackerRotPosition := DINT_TO_USINT(refActionData.aParams[1]);
			CASE eStackerRotPosition OF
				E_StackerRotPosition.LoadingPosition:
					nTurnToPosition := nLoadingPosAngle;
				E_StackerRotPosition.TransferPositionPrinter1:
					nTurnToPosition := nTransferPosAnglePrint1;
				E_StackerRotPosition.TransferPositionPrinter2:
					nTurnToPosition := nTransferPosAnglePrint2;
			ELSE
				M_ExeAction := E_ErrorIdCmd.ERRORID_InvalidStackerAngle;
				RETURN;
			END_CASE
			bTurnTo := TRUE;
		ELSE
			RETURN;
		END_IF
		
	E_Action.ACTION_MoveLifter:
		IF NOT bMoveLifter THEN
			IF NOT P_bTransAreaFree THEN
				M_ExeAction := E_ErrorIdCmd.ERRORID_TransferAreaNotFree;
				RETURN;
			END_IF
			
			IF NOT P_bTraysAligned THEN
				M_ExeAction := E_ErrorIdCmd.ERRORID_TraysNotAligned;
				RETURN;
			END_IF
			
			nMoveLifterPosition := refActionData.aParams[1];
			nMoveLifterSpeed := refActionData.aParams[2];
			bMoveLifter := TRUE;
		ELSE
			RETURN;
		END_IF
		
	E_Action.ACTION_OpenClose:
		IF NOT bOpClTrayStop THEN
			eOpClTrayStopCtrl := DINT_TO_USINT(refActionData.aParams[1]);
			bOpClTrayStop := TRUE;
		ELSE
			RETURN;
		END_IF
		
	E_Action.ACTION_LoadStacker:
		IF NOT P_bTransAreaFree THEN
			M_ExeAction := E_ErrorIdCmd.ERRORID_TransferAreaNotFree;
			RETURN;
		END_IF
		
		IF NOT P_bTraysAligned THEN
			M_ExeAction := E_ErrorIdCmd.ERRORID_TraysNotAligned;
			RETURN;
		END_IF
		
		IF NOT bLoad THEN
			bLoad := TRUE;
		ELSE
			RETURN;
		END_IF
	
END_CASE

eCurrentState := E_MachineState.MACHINESTATE_Active;
bBusy := TRUE;
END_METHOD

METHOD M_GetActionBusy : BOOL
VAR_INPUT
	eAction : E_Action;
END_VAR
CASE eAction OF
	E_Action.ACTION_Init:
		M_GetActionBusy := bInit;
	E_Action.ACTION_TurnTo:
		M_GetActionBusy := bTurnTo;
	E_Action.ACTION_MoveLifter:
		M_GetActionBusy := bMoveLifter;
	E_Action.ACTION_OpenClose:
		M_GetActionBusy := bOpClTrayStop;
	E_Action.ACTION_LoadStacker:
		M_GetActionBusy := bLoad;
END_CASE
END_METHOD

METHOD M_GetAllProps : ERRORID
VAR_INPUT
	refCmdData : REFERENCE TO  ST_CmdData;
END_VAR

VAR
	nCurrentPropIndex	: UINT;
	i : UINT;
END_VAR
refCmdData.aHeader[0] := nObjectID;
refCmdData.aHeader[1] := eObjectType;
refCmdData.aHeader[2]:= nNotifyId;

nCurrentPropIndex := 1;
refCmdData.n32Data[nCurrentPropIndex] := nParentSlotNr;
nCurrentPropIndex := nCurrentPropIndex + 1;
refCmdData.n32Data[nCurrentPropIndex] := nNumberOfShelves;
FOR i := 1 TO nNumberOfShelves DO
	nCurrentPropIndex := nCurrentPropIndex + 1;
	refCmdData.n32Data[nCurrentPropIndex] := aShelfes[i].nPosition;	
END_FOR
nCurrentPropIndex := nCurrentPropIndex + 1;
refCmdData.n32Data[nCurrentPropIndex] := nLoadingPosAngle;
nCurrentPropIndex := nCurrentPropIndex + 1;
refCmdData.n32Data[nCurrentPropIndex] := nTransferPosAnglePrint1;
nCurrentPropIndex := nCurrentPropIndex + 1;
refCmdData.n32Data[nCurrentPropIndex] := nTransferPosAnglePrint2;
END_METHOD

METHOD M_GetBottomShelfPos : DINT
VAR_INPUT
END_VAR

VAR
	i 		: UINT;
	nPos	: DINT;
END_VAR
FOR i := 1 TO nNumberOfShelves DO
	IF aShelfes[i].nPosition > nPos THEN
		nPos :=	aShelfes[i].nPosition;
	END_IF
END_FOR
M_GetBottomShelfPos := nPos;
END_METHOD

METHOD M_GetDevice : I_Device
VAR_INPUT
END_VAR
M_GetDevice := THIS^;
END_METHOD

METHOD M_GetProcData : DINT
VAR_INPUT
	eProcDataType : E_ProcDataType;
END_VAR
END_METHOD

METHOD M_Reset
bBusy := TRUE;
eCurrentState := E_MachineState.MACHINESTATE_Reset;
END_METHOD

METHOD M_SetAllProps : ERRORID
VAR_INPUT
	refCmdData : REFERENCE TO  ST_CmdData;
END_VAR

VAR
	i : UINT;
	nCurrentPropIndex	: UINT;
END_VAR
nCurrentPropIndex := 1;
nParentSlotNr := DINT_TO_UINT(refCmdData.n32Data[nCurrentPropIndex]);
nCurrentPropIndex := nCurrentPropIndex + 1;
//Shelfes (Fächer) parametrieren
nNumberOfShelves := DINT_TO_USINT(refCmdData.n32Data[nCurrentPropIndex]);
IF nNumberOfShelves > cMaxShelfes THEN
	M_SetAllProps := E_ErrorIdObjMgmt.ERRORID_InvalidNumberOfShelfes;
	RETURN;
END_IF

FOR i := 1 TO nNumberOfShelves DO
	nCurrentPropIndex := nCurrentPropIndex + 1;
	aShelfes[i].nPosition := refCmdData.n32Data[nCurrentPropIndex];
	aShelfes[i].bConfigured := TRUE;
END_FOR

{IF defined (Stacker)}
	pHwRef_SpinDrive := ADR(fbHwRefSpinDrive);
	pHwRef_LiftDrive := ADR(fbHwRefLiftDrive);
	pHwRef_TrayStop := ADR(fbHwRefTrayStop);
{ELSE}
	M_SetAllProps := E_ErrorIdObjMgmt.ERRORID_Stacker_NotDefined;
	RETURN;
{END_IF}

nCurrentPropIndex := nCurrentPropIndex + 1;
nLoadingPosAngle := refCmdData.n32Data[nCurrentPropIndex];
nCurrentPropIndex := nCurrentPropIndex + 1;
nTransferPosAnglePrint1 := refCmdData.n32Data[nCurrentPropIndex];
nCurrentPropIndex := nCurrentPropIndex + 1;
nTransferPosAnglePrint2 := refCmdData.n32Data[nCurrentPropIndex];
nNoOfProps := nCurrentPropIndex + 1;
END_METHOD

METHOD M_SetSingleProp : ERRORID
VAR_INPUT
	refCmdData : REFERENCE TO  ST_CmdData;
END_VAR
(*IF nSpecPropIndex = refCmdData.aHeader[1] THEN
	nLoadingPosAngle := refCmdData.n32Data[0];
ELSIF (nSpecPropIndex + 1) = refCmdData.aHeader[1] THEN
	nTransferPosAnglePrint1 := refCmdData.n32Data[0];
ELSIF (nSpecPropIndex + 2) = refCmdData.aHeader[1] THEN
	nTransferPosAnglePrint2 := refCmdData.n32Data[0];
ELSE
	M_SetSingleProp := SUPER^.M_SetSingleProp(refCmdData);
END_IF*)
END_METHOD

METHOD M_Stop : ERRORID
IF eCurrentState = E_MachineState.MACHINESTATE_Active THEN
	IF bInit AND nStateA_Init < 70 THEN
		nStateA_Init := 70;
	END_IF
	
	IF bTurnTo AND nStateA_TurnTo < 70 THEN
		nStateA_TurnTo := 70;
	END_IF
	
	IF bMoveLifter AND nStateA_MoveLifter < 70 THEN
		nStateA_MoveLifter := 70;
	END_IF
	
	IF bOpClTrayStop AND nStateA_OpClTrayStop < 70 THEN
		nStateA_OpClTrayStop := 70;
	END_IF	
END_IF
END_METHOD

PROPERTY P_bBusy : BOOL
GET
P_bBusy := bBusy;
END_GET
END_PROPERTY

PROPERTY P_bCanceled : BOOL
GET
P_bCanceled := bCanceled;
END_GET
END_PROPERTY

PROPERTY P_bError : BOOL
GET
P_bError := (eCurrentState = E_MachineState.MACHINESTATE_Error);
END_GET
END_PROPERTY

PROPERTY P_bIsInit : BOOL
GET
IF pHwRef_SpinDrive > 0 AND_THEN pHwRef_LiftDrive > 0 AND_THEN pHwRef_TrayStop > 0 THEN
	P_bIsInit := pHwRef_SpinDrive^.P_bIsInit AND pHwRef_LiftDrive^.P_bIsInit AND pHwRef_TrayStop^.P_bIsInit;
END_IF
END_GET
SET
bIsInit := P_bIsInit;
END_SET
END_PROPERTY

PROPERTY P_bStopAllOnError : BOOL
GET
P_bStopAllOnError := bStopAllOnError;
END_GET
END_PROPERTY

PROPERTY P_bTransAreaFree : BOOL
GET
P_bTransAreaFree := TRUE;
IF F_GetMappingStatus(ADR(bSensorTransAreaLeft),SIZEOF(bSensorTransAreaLeft)) = EPlcMappingStatus.MS_Partial THEN
	IF NOT bSensorTransAreaLeft THEN
		P_bTransAreaFree := FALSE;
	END_IF
END_IF

IF F_GetMappingStatus(ADR(bSensorTransAreaRight),SIZEOF(bSensorTransAreaRight)) = EPlcMappingStatus.MS_Partial THEN
	IF NOT bSensorTransAreaRight THEN
		P_bTransAreaFree := FALSE;
	END_IF	
END_IF
END_GET
END_PROPERTY

PROPERTY P_bTrayInCurrentShelf : BOOL
GET
P_bTrayInCurrentShelf := bSensorTrayDetection;
END_GET
END_PROPERTY

PROPERTY P_bTraysAligned : BOOL
GET
P_bTraysAligned := bSensorTrayAlignmentLeft AND bSensorTrayAlignmentRight;
END_GET
END_PROPERTY

PROPERTY P_eCurrentSpinPositon : E_StackerRotPosition
GET
VAR
	nActPosTemp : DINT;
END_VAR
IF pHwRef_SpinDrive^.P_nActualPosition > 359000 THEN
	nActPosTemp := -(360000 - pHwRef_SpinDrive^.P_nActualPosition);
ELSE
	nActPosTemp := pHwRef_SpinDrive^.P_nActualPosition;
END_IF

IF nActPosTemp >= (nLoadingPosAngle - 100) AND nActPosTemp <= (nLoadingPosAngle + 100) THEN
	P_eCurrentSpinPositon := E_StackerRotPosition.LoadingPosition;
ELSIF nActPosTemp >= (nTransferPosAnglePrint1 - 100) AND nActPosTemp <= (nTransferPosAnglePrint1 + 100) THEN
	P_eCurrentSpinPositon := E_StackerRotPosition.TransferPositionPrinter1;
ELSIF nActPosTemp >= (nTransferPosAnglePrint2 - 100) AND nActPosTemp <= (nTransferPosAnglePrint2 + 100) THEN
	P_eCurrentSpinPositon := E_StackerRotPosition.TransferPositionPrinter2;
ELSE
	P_eCurrentSpinPositon := E_StackerRotPosition.UNDEFINED;
END_IF
END_GET
END_PROPERTY

PROPERTY P_eCurrentState : E_MachineState
GET
P_eCurrentState := eCurrentState;
END_GET
END_PROPERTY

PROPERTY P_nCurrentShelf : UINT
GET
VAR
	i : USINT;
END_VAR
FOR i := 1 TO nNumberOfShelves DO
	IF pHwRef_LiftDrive^.P_nActualPosition >= aShelfes[i].nPosition - 200 AND pHwRef_LiftDrive^.P_nActualPosition <= aShelfes[i].nPosition + 200 THEN
		P_nCurrentShelf := i;
		EXIT;
	END_IF
END_FOR
END_GET
END_PROPERTY

PROPERTY P_nErrorId : ERRORID
GET
P_nErrorID := stError.ErrorId;
END_GET
END_PROPERTY

PROPERTY P_nNotifyId : UINT
GET
P_nNotifyId := nNotifyId;
END_GET
SET
nNotifyId := P_nNotifyId;
END_SET
END_PROPERTY

PROPERTY P_nParentSlotNr : UINT
GET
P_nParentSlotNr := nParentSlotNr;
END_GET
END_PROPERTY

PROPERTY P_pObject : POINTER TO FB_Object
GET
P_pObject := THIS;
END_GET
END_PROPERTY

PROPERTY P_stError : ST_Error
GET
END_GET
END_PROPERTY

END_FUNCTION_BLOCK

// ---- Hardware/EL70xxDrive/FB_HwRefEL70xxDrive.TcPOU
FUNCTION_BLOCK FB_HwRefEL70xxDrive EXTENDS FB_HwModule
VAR_INPUT
	STM_Control : ST_EL70xx_STM_Control;
	POS_Control	: ST_EL70xx_POS_Control;	
END_VAR
VAR_OUTPUT
	STM_Status : ST_EL70xx_STM_Status;
	POS_Status : ST_EL70xx_POS_Status;
	nMotorLoad 		AT %I* : UINT;
	nMotorCurrent 	AT %I* : UINT;
	bInput1			AT %I* : BOOL;
	bInput2			AT %I* : BOOL;
	bHwEnable		AT %I* : BOOL;	//muss mit Input1 oder Input2 der Klemme verknüpft werden
									//entsprechend muss dieser Input auch konfiguriert werden
									//8012:32 bzw. 36 auf Hardware enable konfigurieren
	
END_VAR
VAR
	stAdsAddress : ST_AdsAdress;	
	rTranslationFactorPosition : REAL;
	
	fbEcCoESdoRead 			: FB_EcCoESdoRead;
	nMotorFullsteps 		: UINT;
	nEncoderIncrements		: UDINT;
	nSpeedRangeRaw			: USINT;	//wie es im OD steht
	nSpeedRangeCalculated	: UINT;		//wird berechnet aus 2^nSpeedRangeRaw * 1000
	eEncoderType			: E_EL70xx_EncoderType := E_EL70xx_EncoderType.InternCounter;
	sTermName				: STRING(5);
	
	nActualPosition			: DINT;
	eHomingMode				: E_EL70xx_StartType;
	bPrepare				: BOOL;
	nStateA_Prepare 		: USINT;
	
END_VAR
VAR PERSISTENT
	nDistPerMotorRev	: DINT; //reale Einheit (Weg oder Winkel)
	nRefPos	 			: DINT; //reale Einheit (Weg oder Winkel)
	nMinPos				: DINT; //reale Einheit (Weg oder Winkel)
	nMaxPos				: DINT; //reale Einheit (Weg oder Winkel)
	nMaxSpeed			: DINT;	//reale Einheit/s
	bInvertInitDir		: BOOL;
END_VAR

IF bPrepare THEN
	bBusy := TRUE;
	A_Prepare();
	IF nStateA_Prepare >= 80 THEN
		IF nStateA_Prepare >= 99 THEN
			bError := TRUE;
		END_IF
		nStateA_Prepare := 0;
		bPrepare := FALSE;
		bBusy := FALSE;
	END_IF
ELSE
	bBusy := POS_Status.Busy;
	bError := POS_Status.Error OR STM_Status.Error;
	A_CalcActPosition();
END_IF

ACTION A_CalcActPosition:
IF rTranslationFactorPosition > 0 THEN
	nActualPosition := REAL_TO_DINT(DINT_TO_REAL(POS_Status.ActualPosition) / rTranslationFactorPosition);
END_IF
END_ACTION

ACTION A_Prepare:
//Werte aus Coe auslesen
//Motor fullsteps (8010:06)
IF nStateA_Prepare = 0 THEN
	fbEcCoESdoRead(sNetId:= stAdsAddress.sNetId, nSlaveAddr:= stAdsAddress.nPort, nIndex:= 16#8010, nSubIndex:= 6 , 
					pDstBuf:= ADR(nMotorFullsteps) , cbBufLen:=SIZEOF(nMotorFullsteps) , bExecute:= TRUE);
	IF NOT fbEcCoESdoRead.bBusy THEN
		IF fbEcCoESdoRead.bError THEN
			nStateA_Prepare := 99;
		ELSE
			IF eEncoderType <> E_EL70xx_EncoderType.InternCounter THEN //Initialwert
				//Encodertype wurde bereits in der abgeleiteten Klasse gesetzt, deshalb wird dieser nicht aus der Klemme gelesen
				//auch die Inkremente werden nicht gelesen, diese werden auch in der abgeleiteten Klasse gesetzt
				nStateA_Prepare := 3;
			ELSE
				nStateA_Prepare := 1;	
			END_IF			
		END_IF
		fbEcCoESdoRead(bExecute:= FALSE);		
	END_IF
END_IF
 
//die ersten 5 Stellen des Klemmentyps auslesen
IF nStateA_Prepare = 1 THEN
	fbEcCoESdoRead(nIndex:= 16#1008, nSubIndex:= 0, pDstBuf:= ADR(sTermName), cbBufLen:=SIZEOF(sTermName), bExecute:= TRUE);
	IF NOT fbEcCoESdoRead.bBusy THEN
		IF fbEcCoESdoRead.bError THEN
			nStateA_Prepare := 99;
		ELSE
			sTermName[5] := 0; //da der String nicht komplett ausgelesen wurde, muss das letzte Byte im String wieder terminiert werden
			IF sTermName = 'EL704' THEN //nur die Klemmen dieser Reihe können einen internen Encoder
				nStateA_Prepare := 2;
			ELSE
				nStateA_Prepare := 4;
			END_IF
		END_IF
		fbEcCoESdoRead(bExecute:= FALSE);
	END_IF
END_IF

//Encodertype bzw. Feedback auslesen (8012:08)
IF nStateA_Prepare = 2 THEN
	fbEcCoESdoRead(nIndex:= 16#8012, nSubIndex:= 8, pDstBuf:= ADR(eEncoderType) , cbBufLen:=SIZEOF(eEncoderType), bExecute:= TRUE);
	IF NOT fbEcCoESdoRead.bBusy THEN
		IF fbEcCoESdoRead.bError THEN
			nStateA_Prepare := 99;	
		ELSE
			IF eEncoderType = E_EL70xx_EncoderType.InternEncoder THEN
				nStateA_Prepare := 3;
			ELSE
				nStateA_Prepare := 4;
			END_IF
		END_IF
		fbEcCoESdoRead(bExecute:= FALSE);
	END_IF	
END_IF

//Encoder increments (8010:07) nur wenn Feedbacktype "InternEncoder"
//Achtung, nEncoderIncrements ist UDINT, der Wert im OD aber nur UINT
IF nStateA_Prepare = 3 THEN
	fbEcCoESdoRead(nIndex:= 16#8010, nSubIndex:= 7, pDstBuf:= ADR(nEncoderIncrements) , cbBufLen:= 2, bExecute:= TRUE);
	IF NOT fbEcCoESdoRead.bBusy THEN
		IF fbEcCoESdoRead.bError THEN
			nStateA_Prepare := 99;
		ELSE
			nStateA_Prepare := 4;
		END_IF
		fbEcCoESdoRead(bExecute:= FALSE);		
	END_IF	
END_IF

//Speedrange (8012:05)
IF nStateA_Prepare = 4 THEN
	fbEcCoESdoRead(nIndex:= 16#8012, nSubIndex:= 5, pDstBuf:= ADR(nSpeedRangeRaw) , cbBufLen:=SIZEOF(nSpeedRangeRaw), bExecute:= TRUE);
	IF NOT fbEcCoESdoRead.bBusy THEN
		IF fbEcCoESdoRead.bError THEN
			nStateA_Prepare := 99;	
		ELSE
			nSpeedRangeCalculated := SHL(1,nSpeedRangeRaw) * 1000;
			M_CalcTranslationFact();
			nStateA_Prepare := 80;
		END_IF
		fbEcCoESdoRead(bExecute:= FALSE);		
	END_IF	
END_IF
END_ACTION

METHOD FB_init : BOOL
VAR_INPUT
	bInitRetains 	: BOOL; 	// if TRUE, the retain variables are initialized (warm start / cold start)
	bInCopyCode  	: BOOL;  	// if TRUE, the instance afterwards gets moved into the copy code (online change)
	nBoxAddress		: UINT;
	eHomingMode		: E_EL70xx_StartType;
END_VAR

VAR
END_VAR
THIS^.eHomingMode := eHomingMode;
stAdsAddress.nPort := nBoxAddress;
END_METHOD

METHOD M_CalcTranslationFact
VAR_INPUT
END_VAR
IF nDistPerMotorRev > 0 THEN
	IF eEncoderType = E_EL70xx_EncoderType.InternCounter OR eEncoderType = E_EL70xx_EncoderType.ExternSingleturnAbs THEN 
		rTranslationFactorPosition := (nMotorFullsteps * 64) / DINT_TO_REAL(nDistPerMotorRev);
	ELSE
		rTranslationFactorPosition := UDINT_TO_REAL(nEncoderIncrements) / DINT_TO_REAL(nDistPerMotorRev);
	END_IF
END_IF
END_METHOD

METHOD M_GetPosDiff : DINT
VAR_INPUT
	nSetPosition : DINT;
END_VAR
M_GetPosDiff := nSetPosition - P_nActualPosition;
END_METHOD

METHOD M_Prepare
VAR_INPUT
END_VAR
bPrepare := TRUE;
END_METHOD

METHOD M_SetSpeed : BOOL
VAR_INPUT
	nValue : DINT; //Speed in µm/s oder 1/100°/sec
END_VAR
IF (nValue > 0) AND (nValue <= nMaxSpeed) THEN
	POS_Control.Velocity := DINT_TO_INT(nMotorFullsteps * nValue / nDistPerMotorRev * 10000 / nSpeedRangeCalculated);
	M_SetSpeed := TRUE;
END_IF
END_METHOD

METHOD M_SetTargetPos : BOOL
VAR_INPUT
	nValue : DINT; //Reale Einheit
END_VAR
IF (nValue >= nMinPos) AND (nValue <= nMaxPos) THEN
	POS_Control.StartType := E_EL70xx_StartType.Absolute;
	POS_Control.TargetPosition := REAL_TO_DINT(DINT_TO_REAL(nValue) * rTranslationFactorPosition);
	M_SetTargetPos := TRUE;
END_IF
END_METHOD

PROPERTY P_bHardwareEnable : BOOL
GET
IF F_GetMappingStatus(ADR(bHwEnable), SIZEOF(bHwEnable)) = EPlcMappingStatus.MS_Partial THEN
	P_bHardwareEnable := bHwEnable;
ELSE
	P_bHardwareEnable := TRUE;
END_IF
END_GET
END_PROPERTY

PROPERTY P_bInvertInitDir : BOOL
GET
P_bInvertInitDir := bInvertInitDir;
END_GET
SET
bInvertInitDir := P_bInvertInitDir;
fbSettings.M_WritePersData();
END_SET
END_PROPERTY

PROPERTY P_bIsInit : BOOL
GET
P_bIsInit := POS_Status.Calibrated;
END_GET
END_PROPERTY

PROPERTY P_eEncoderType : E_EL70xx_EncoderType
GET
P_eEncoderType := eEncoderType;
END_GET
END_PROPERTY

PROPERTY P_eHomingMode : E_EL70xx_StartType
GET
P_eHomingMode := eHomingMode;
END_GET
END_PROPERTY

PROPERTY P_nActualPosition : DINT
GET
A_CalcActPosition();
P_nActualPosition := nActualPosition;
END_GET
END_PROPERTY

PROPERTY P_nDistPerMotorRev : DINT
GET
P_nDistPerMotorRev := nDistPerMotorRev;
END_GET
SET
nDistPerMotorRev := P_nDistPerMotorRev;
M_CalcTranslationFact();
fbSettings.M_WritePersData();
END_SET
END_PROPERTY

PROPERTY P_nMaxPos : DINT
GET
P_nMaxPos := nMaxPos;
END_GET
SET
nMaxPos := P_nMaxPos;
fbSettings.M_WritePersData();
END_SET
END_PROPERTY

PROPERTY P_nMaxSpeed : DINT
GET
P_nMaxSpeed := nMaxSpeed;
END_GET
SET
nMaxSpeed := P_nMaxSpeed;
fbSettings.M_WritePersData();
END_SET
END_PROPERTY

PROPERTY P_nMinPos : DINT
GET
P_nMinPos := nMinPos;
END_GET
SET
nMinPos := P_nMinPos;
fbSettings.M_WritePersData();
END_SET
END_PROPERTY

PROPERTY P_nRefPos : DINT
GET
P_nRefPos := nRefPos;
END_GET
SET
nRefPos := P_nRefPos;
fbSettings.M_WritePersData();
END_SET
END_PROPERTY

PROPERTY P_nRefPosRaw : DINT
GET
P_nRefPosRaw := REAL_TO_DINT(DINT_TO_REAL(nRefPos) * rTranslationFactorPosition);
END_GET
END_PROPERTY

PROPERTY P_nSlaveAddr : UINT
GET
P_nSlaveAddr := stAdsAddress.nPort;
END_GET
END_PROPERTY

PROPERTY P_sNetId : STRING(23)
GET
P_sNetId := stAdsAddress.sNetId;
END_GET
SET
stAdsAddress.sNetId := P_sNetId;
END_SET
END_PROPERTY

END_FUNCTION_BLOCK

// ---- Hardware/EL70xxDrive/FB_HWECtrl_EL70xx_Power.TcPOU
FUNCTION_BLOCK FB_HWECtrl_EL70xx_Power
VAR_INPUT
	bExecute	: BOOL;
	bEnable		: BOOL;
END_VAR
VAR_OUTPUT
	bBusy 		: BOOL;
	bError 		: BOOL;
	nErrorId 	: ERRORID;		
END_VAR
VAR_IN_OUT
	pHwRef : POINTER TO FB_HwRefEL70xxDrive; 
END_VAR
VAR
	nState 	: USINT;
	timer	: TON;
END_VAR

IF bExecute THEN
	IF nState = 0 THEN
		IF bEnable THEN
			IF pHwRef^.P_bHardwareEnable THEN
				nState := 1;
			ELSE
				nErrorId := E_ErrorIdHwGeneral.ERRORID_HardwareNotEnabled;
				bError := TRUE;
				nState := 99;
				RETURN;
			END_IF
		ELSE
			nState := 2;
		END_IF
	END_IF

	IF nState = 1 THEN //Enable
		IF pHwRef^.STM_Status.Error OR pHwRef^.POS_Status.Error THEN
			bBusy := TRUE;
			pHwRef^.STM_Control.Reset := TRUE;
		ELSIF pHwRef^.STM_Status.Ready THEN
			pHwRef^.STM_Control.ReduceTorque := TRUE;
			pHwRef^.STM_Control.Reset := FALSE;
			bBusy := FALSE;
			RETURN;
		ELSIF pHwRef^.STM_Status.ReadyToEnable THEN
			bBusy := TRUE;
			pHwRef^.STM_Control.Reset := FALSE;
			pHwRef^.STM_Control.Enable := TRUE;
		END_IF
		timer(IN:= TRUE, PT:= T#5000MS);
		IF timer.Q AND bBusy THEN
			timer(IN:= FALSE);
			nErrorId := E_ErrorIdHwGeneral.ERRORID_Timeout;
			bBusy := FALSE;
			bError := TRUE;
			nState := 99;
		END_IF
	ELSIF nState = 2 THEN //Disable
		pHwRef^.STM_Control.Enable := FALSE;
		bBusy := FALSE;
	END_IF
ELSE
	timer(IN:= FALSE);
	bBusy := FALSE;
	bError := FALSE;
	bEnable := FALSE;
	nState := 0;	
END_IF

END_FUNCTION_BLOCK

// ---- Hardware/EL70xxDrive/FB_HWECtrl_EL70xx_Home.TcPOU
FUNCTION_BLOCK FB_HWECtrl_EL70xx_Home
VAR_INPUT
	bExecute : BOOL;
	bStop	 : BOOL;
END_VAR
VAR_OUTPUT
	bBusy 		: BOOL;
	bError 		: BOOL;
	nErrorId 	: ERRORID;		
END_VAR
VAR_IN_OUT
	pHwRef : POINTER TO FB_HwRefEL70xxDrive; 
END_VAR
VAR
	nState 			: USINT;
	nData32 		: DINT;
	nDataBool		: BOOL;
	fbEcCoESdoWrite : FB_EcCoESdoWrite;
END_VAR

IF bExecute THEN
	CASE nState OF
		0:	//Home position in Klemme schreiben
			bBusy := TRUE;
			nData32 := pHwRef^.P_nRefPosRaw;
			fbEcCoESdoWrite(sNetId:= pHwRef^.P_sNetId, nSlaveAddr:= pHwRef^.P_nSlaveAddr,
				nIndex:=16#8020, nSubIndex:= 16#08, pSrcBuf:=ADR(nData32) ,cbBufLen:= SIZEOF(nData32), bExecute:= TRUE);
			IF NOT fbEcCoESdoWrite.bBusy THEN
				IF fbEcCoESdoWrite.bError THEN
					nErrorId := UDINT_TO_UINT(fbEcCoESdoWrite.nErrId);
					nState := 99;
				ELSE
					nState := 1;
				END_IF
				fbEcCoESdoWrite(bExecute:= FALSE);
			END_IF
			
		1:	//Init direction in Klemme schreiben Teil 1 (Invert calibration cam search direction)
			nDataBool := NOT pHwRef^.P_bInvertInitDir;
			fbEcCoESdoWrite(nIndex:=16#8021, nSubIndex:= 16#13, pSrcBuf:=ADR(nDataBool) ,cbBufLen:= SIZEOF(nDataBool), bExecute:= TRUE);
			IF NOT fbEcCoESdoWrite.bBusy THEN
				IF fbEcCoESdoWrite.bError THEN
					nErrorId := UDINT_TO_UINT(fbEcCoESdoWrite.nErrId);
					nState := 99;
				ELSE
					nState := 2;
				END_IF
				fbEcCoESdoWrite(bExecute:= FALSE);
			END_IF
			
		2:	//Init direction in Klemme schreiben Teil 2 (Invert sync impulse search direction)
			nDataBool := pHwRef^.P_bInvertInitDir;
			fbEcCoESdoWrite(nIndex:=16#8021, nSubIndex:= 16#14, pSrcBuf:=ADR(nDataBool) ,cbBufLen:= SIZEOF(nDataBool), bExecute:= TRUE);
			IF NOT fbEcCoESdoWrite.bBusy THEN
				IF fbEcCoESdoWrite.bError THEN
					nErrorId := UDINT_TO_UINT(fbEcCoESdoWrite.nErrId);
					nState := 99;
				ELSE
					nState := 3;
				END_IF
				fbEcCoESdoWrite(bExecute:= FALSE);
			END_IF
			
		3:	//Homing Mode setzen
			//Homing Position setzen
			IF bStop THEN
				nState := 80;	
			ELSE
				pHwRef^.POS_Control.StartType := pHwRef^.P_eHomingMode;
				pHwRef^.STM_Control.ReduceTorque := FALSE;
				pHwRef^.POS_Control.Execute := TRUE;
				nState := 4;
			END_IF
			
		4:	IF pHwRef^.POS_Status.Busy OR bStop THEN
				nState := 5;
			END_IF
			
		5:	IF bStop THEN
				pHwRef^.POS_Control.Execute := FALSE;
				nState := 6;
			ELSE
				IF NOT pHwRef^.POS_Status.Busy THEN
					IF pHwRef^.POS_Status.Calibrated THEN
						nState := 80;
					ELSE
						nErrorId := E_ErrorIdHwGeneral.ERRORID_HomingFailed;
						nState := 99;
					END_IF
				ELSIF pHwRef^.POS_Status.Error THEN
					nErrorId := E_ErrorIdHwGeneral.ERRORID_HomingFailed;
					nState := 99;
				END_IF
			END_IF
			
		6:	//es wurde gestoppt
			IF NOT pHwRef^.POS_Status.Busy THEN
				nState := 80;
			END_IF		
			
	END_CASE
	
	IF nState >= 80 THEN
		pHwRef^.POS_Control.Execute := FALSE;
		pHwRef^.STM_Control.ReduceTorque := TRUE;
		IF nState = 99 THEN
			bError := TRUE;	
		END_IF
		bBusy := FALSE;
	END_IF

ELSE
	bBusy := FALSE;
	bError := FALSE;
	nErrorId := 0;
	nState := 0;	
END_IF

END_FUNCTION_BLOCK

// ---- Hardware/EL70xxDrive/FB_HWECtrl_EL70xx_Move.TcPOU
FUNCTION_BLOCK FB_HWECtrl_EL70xx_Move
VAR_INPUT
	bExecute			: BOOL;
	bStop				: BOOL;
	nPosition			: DINT;	//Reale Einheit (µm oder µ°)
	nSpeed				: DINT;	//Reale Einheit/s
	nToleranceWindow 	: DINT;	//in diesem Bereich muss am Ende die Position liegen, wenn nicht, dann wird ein Fehler geworfen
								//wenn ToleranceWindow auf 0 steht, dann wird nicht überwacht 
END_VAR
VAR_OUTPUT
	bBusy 		: BOOL;
	bError 		: BOOL;
	nErrorId 	: ERRORID;		
END_VAR
VAR_IN_OUT
	pHwRef : POINTER TO FB_HwRefEL70xxDrive; 
END_VAR
VAR
	nState 			: USINT;
	nReadjustments 	: USINT;
	nPosDiffernce	: DINT;
END_VAR

IF bExecute THEN
	//Vorbedingungen prüfen
	IF nState = 0 THEN
		nState := 1;
		
		IF pHwRef^.bError THEN
			{warning 'Implement}
			nErrorID := 8145;
			nState := 99;
		END_IF
		
		IF pHwRef^.bBusy THEN
			{warning 'Implement}
			nErrorID := 8146;
			nState := 99;
		END_IF
		
		IF NOT pHwRef^.P_bIsInit THEN
			nErrorID := E_ErrorIdHwGeneral.ERRORID_DriveNotHomed;
			nState := 99;
		END_IF
		
		IF NOT pHwRef^.M_SetTargetPos(nPosition) THEN
			nErrorID := E_ErrorIdHwGeneral.ERRORID_InvalidPosition;
			nState := 99;
		END_IF
		
		IF  NOT pHwRef^.M_SetSpeed(nSpeed) THEN
			nErrorID := E_ErrorIdHwGeneral.ERRORID_InvalidSpeed;
			nState := 99;
		END_IF
	END_IF

	CASE nState OF
		1:	//Starttype schreiben
			bBusy := TRUE;
			IF bStop THEN
				nState := 80;
			ELSE
				pHwRef^.POS_Control.Execute := TRUE;
				pHwRef^.STM_Control.ReduceTorque := FALSE;
				nState := 2;
			END_IF

		2:	//Warten auf Busy
			IF bError THEN
				nErrorID := E_ErrorIdHwGeneral.ERRORID_UndefinedDriveError;
				nState := 99;
			ELSE
				IF bStop THEN
					pHwRef^.POS_Control.Execute := FALSE;
					nState := 4;
				ELSE
					IF pHwRef^.POS_Status.Busy THEN
						nState := 3;
					END_IF
				END_IF
			END_IF

		3:	IF bStop THEN
				pHwRef^.POS_Control.Execute := FALSE;
				nState := 4;
			ELSE
				IF NOT pHwRef^.POS_Status.Busy THEN
					IF pHwRef^.POS_Status.Error OR pHwRef^.STM_Status.Error THEN
						IF NOT pHwRef^.P_bHardwareEnable THEN
							nErrorID := E_ErrorIdHwGeneral.ERRORID_HardwareNotEnabled;
						ELSE
							nErrorID := E_ErrorIdHwGeneral.ERRORID_UndefinedDriveError;
						END_IF
						pHwRef^.POS_Control.Execute := FALSE;
						nState := 99;
					ELSE
						//InTarget?
						IF pHwRef^.POS_Status.InTarget THEN
							pHwRef^.POS_Control.Execute := FALSE;
							nPosDiffernce := ABS(pHwRef^.M_GetPosDiff(nPosition));
							nState := 80;
							IF nToleranceWindow > 0 AND_THEN nPosDiffernce > nToleranceWindow THEN
								IF pHwRef^.P_eEncoderType = E_EL70xx_EncoderType.ExternSingleturnAbs AND_THEN nReadjustments < 3 THEN //nachjustieren
									nReadjustments := nReadjustments + 1;
									nState := 0;
								ELSE
									//Positionierung war nicht im zulässigen Toleranzbereich
									nErrorID := E_ErrorIdHwGeneral.ERRORID_PosOutsideToleranceWindow;
									nState := 99;
								END_IF
							END_IF
						ELSE
							pHwRef^.POS_Control.Execute := FALSE;
							nErrorID := E_ErrorIdHwGeneral.ERRORID_TargetPosNotReached;
							nState := 99;
						END_IF
					END_IF
				END_IF
			END_IF
			
		4:	//Warten bis gestoppt
			IF NOT pHwRef^.POS_Status.Busy THEN
				nState := 80;
			END_IF		
	END_CASE
	
	IF nState >= 80 THEN
		pHwRef^.STM_Control.ReduceTorque := TRUE;
		IF nState = 99 THEN
			bError := TRUE;	
		END_IF
		bBusy := FALSE;
	END_IF

ELSE
	bBusy := FALSE;
	bError := FALSE;
	bStop := FALSE;
	nErrorId := 0;
	nState := 0;
	nReadjustments := 0;	
END_IF

END_FUNCTION_BLOCK

// ---- Configuration/FB_Configuration.TcPOU
FUNCTION_BLOCK FB_Configuration
VAR_INPUT
	bExecute : BOOL;
END_VAR
VAR_OUTPUT
	bError : BOOL;
	bBusy : BOOL;
	nErrorId : ERRORID;
	stError	: ST_Error;
END_VAR
VAR
	//Diese beiden Variablen müssen hintereinander stehen !!////
	nBytesNextRead : UINT;
	///////////////////////////////////////////////////////////
	bActivated : BOOL;
	bActivate : BOOL;
	nStateA_Activate 	: USINT;
	pMultiZRef	: POINTER TO FB_MultiZRef;
	
	//Load/Save
	fbFileOpen		: FB_FileOpen;
	fbFileClose		: FB_FileClose;
	fbFileWrite		: FB_FileWrite;
	fbFileRead		: FB_FileRead;
	fbFileDelete	: FB_FileDelete;
	hFile			: UINT;
	//Diese beiden Variablen müssen hintereinander stehen !!////
	nBytesWrite		: UINT;
	stPropData		: ST_CmdData;
	///////////////////////////////////////////////////////////
	
	nStateA_LoadSaveDel : USINT;
	
	nCheckObjPropsObjId	: UINT;
	nCheckObjPropsObjIdStart: UINT;
	nCheckObjCount : UINT;
	timer : TON;
	pObject : POINTER TO FB_Object;
	iter	: FB_ObjCollectIteratorDeep;
END_VAR
VAR CONSTANT
	sConfigPath	: STRING := '\Hard Disk\TwinCAT\3.1\Boot\Standard.cfg';
END_VAR
VAR PERSISTENT
	bConfigSaved : BOOL;
END_VAR

ACTION A_Delete:
IF bExecute THEN
	bBusy := TRUE;
	bConfigSaved := FALSE;
	fbSettings.M_WritePersData();
	fbFileDelete(sPathName:= sConfigPath, bExecute:= TRUE);
	IF NOT fbFileDelete.bBusy THEN
		IF fbFileDelete.bError THEN
			bError := TRUE;
		END_IF
		fbFileDelete(bExecute:= FALSE);
		bBusy := FALSE;
	END_IF
ELSE
	bError := FALSE;	
END_IF
END_ACTION

ACTION A_Activate:

IF bExecute THEN
	//**************************Begin CheckObjects**********************************
	IF nStateA_Activate = 0 THEN
		bActivated := FALSE;
		//Es ist mindestens ein Head und eine Workplate zum aktivieren erforderlich
		IF fbObjectDirectory.nCntMZHead = 0 THEN
			stError.ErrorId := E_ErrorIdObjMgmt.ERRORID_NoHeadCreated;
			bError := TRUE;
			RETURN;
		END_IF
		
		IF fbObjectDirectory.nCntWorkplate = 0 THEN
			stError.ErrorId := E_ErrorIdObjMgmt.ERRORID_NoWorkplateCreated;
			bError := TRUE;
			RETURN;
		END_IF
		
		bBusy := TRUE;
		
		nCheckObjPropsObjIdStart := 1;
		nStateA_Activate := 1;
		fbObjectDirectory.P_pDeviceCollection^.M_GetIterator(iter);
	END_IF
	
	IF nStateA_Activate = 1 THEN
		//Es werden max. 100 Objekte in einem Zyklus gecheckt
		//Achtung, hier besteht die Gefahr, dass die ObjectIDs nicht in der Reihenfolge sind
		nCheckObjCount := 0;
		WHILE iter.pNode > 0 AND_THEN iter.pNode^.P_pObject > 0 DO
			nCheckObjCount := nCheckObjCount + 1;
			pObject := iter.pNode^.P_pObject;
			stError.ObjectId := pObject^.P_nObjectID;
			stError.ErrorId := pObject^.M_CheckProps();
			IF stError.ErrorId > 0 THEN
				nStateA_Activate := 99;
				EXIT;
			ELSE
				IF nCheckObjCount = 100 THEN
					RETURN;
				ELSE
					nStateA_Activate := 20;
				END_IF
			END_IF
			iter.M_Increment();
		END_WHILE
	END_IF
	//***************************End CheckObjects***********************************
	//***************************Begin ResetMzBase**********************************
	IF nStateA_Activate = 10 THEN
		fbMultiZRefList.M_SetCurrentToHead();
		REPEAT
			pMultiZRef := fbMultiZRefList.M_Get();
			IF pMultiZRef > 0 THEN
				pMultiZRef^.M_Reset();
			END_IF
		UNTIL pMultiZRef = 0
		END_REPEAT
		nStateA_Activate := 11;
	END_IF
	
	IF nStateA_Activate = 11 THEN
		nStateA_Activate := 20;
		fbMultiZRefList.M_SetCurrentToHead();
		REPEAT
			pMultiZRef := fbMultiZRefList.M_Get();
			IF pMultiZRef > 0 THEN
				IF pMultiZRef^.bBusy THEN
					nStateA_Activate := 11;	
				END_IF
				IF pMultiZRef^.bError THEN
					nStateA_Activate := 99;
				END_IF
			END_IF
		UNTIL pMultiZRef = 0
		END_REPEAT
	END_IF
	//****************************End ResetMzBase***********************************
	//**************************Begin Set MzConfig***********************************
	IF nStateA_Activate = 20 THEN
		fbMultiZRefList.M_SetCurrentToHead();
		REPEAT
			pMultiZRef := fbMultiZRefList.M_Get();
			IF pMultiZRef > 0 THEN
				pMultiZRef^.M_SetConfig();
			END_IF
		UNTIL pMultiZRef = 0
		END_REPEAT
		nStateA_Activate := 21;	
	ELSIF nStateA_Activate = 21 THEN
		nStateA_Activate := 80;
		fbMultiZRefList.M_SetCurrentToHead();
		REPEAT
			pMultiZRef := fbMultiZRefList.M_Get();
			IF pMultiZRef > 0 THEN
				IF pMultiZRef^.bBusy THEN
					nStateA_Activate := 21;
				END_IF
				IF pMultiZRef^.bError THEN
					stError := pMultiZRef^.P_stError;
					stError.POU := E_POU.POU_FB_Configuration;
					stError.POUAction := E_POUACT.POUACT_A_Activate;
					nStateA_Activate := 99;
				END_IF
			END_IF
		UNTIL pMultiZRef = 0
		END_REPEAT
	END_IF
	//***************************End Set MzConfig************************************
	
	
	//Nur zum debuggen
	IF nStateA_Activate = 30 THEN
		timer(IN:= TRUE,PT:=T#10S);
		IF timer.Q THEN
			timer(IN:= FALSE);
			nStateA_Activate := 80;
		END_IF
	END_IF
	
	IF nStateA_Activate = 80 THEN
		bBusy := FALSE;
		bActivated := TRUE;
	ELSIF nStateA_Activate = 99 THEN
		bError := TRUE;
		bBusy := FALSE;
	END_IF
ELSE
	nStateA_Activate := 0;
	bError := FALSE;
END_IF
END_ACTION

ACTION A_Save:
IF bExecute THEN
	IF nStateA_LoadSaveDel = 0 THEN //File "Standard.cfg" zum schreiben öffnen
		bBusy := TRUE;
		hFile := 0;
		fbFileOpen(sPathName:= sConfigPath, nMode:= FOPEN_MODEWRITE OR FOPEN_MODEBINARY, bExecute:= TRUE);
		IF NOT fbFileOpen.bBusy THEN
			IF fbFileOpen.bError THEN
				nErrorId := UDINT_TO_UINT(fbFileOpen.nErrId);
				nStateA_LoadSaveDel := 99;
			ELSE
				hFile := fbFileOpen.hFile;
				fbObjectDirectory.P_pObjectCollection^.M_GetIterator(iter);
				nStateA_LoadSaveDel := 2;
			END_IF
			fbFileOpen(bExecute:= FALSE);
		END_IF
	END_IF
	
	IF nStateA_LoadSaveDel = 2 THEN
		//Alle Objekte durchlaufen -> M_GetAllProps
		IF NOT fbFileWrite.bBusy AND iter.pNode > 0 AND_THEN iter.pNode^.P_pObject > 0 THEN
			pObject := iter.pNode^.P_pObject;
			MEMSET(ADR(stPropData),0,SIZEOF(stPropData));
			pObject^.M_GetAllProps(refCmdData:= stPropData);
			nBytesWrite := 2 + 8 + pObject^.P_nNoOfProps * 4;
			iter.M_Increment();
		END_IF
		//File wird im binary-format geschieben
		//Aufbau des Files:
		//Objekte
		//nBytesWrite(2Byte) ; ObjectHeader: Header[0]ObjectId(2Byte) ; Header[1]ObjectType(2Byte) ; Header[2]n.a(2Byte) ; Header[3]n.a(2Byte) ; Data[0](4Btye) ; usw
		fbFileWrite(hFile:= hFile, pWriteBuff:= ADR(nBytesWrite), cbWriteLen:= nBytesWrite, bExecute:= TRUE);
		IF NOT fbFileWrite.bBusy THEN
			IF fbFileWrite.bError THEN
				nErrorId := UDINT_TO_UINT(fbFileWrite.nErrId);
				nStateA_LoadSaveDel := 99;				
			ELSE
				fbFileWrite(bExecute:= FALSE);
				IF iter.pNode = 0 THEN
					nStateA_LoadSaveDel := 3;
				END_IF
			END_IF
		END_IF
	END_IF
	
	IF nStateA_LoadSaveDel = 3 OR nStateA_LoadSaveDel = 99 THEN
		IF hFile > 0 THEN
			fbFileClose(hFile:= hFile, bExecute:= TRUE);
			IF NOT fbFileClose.bBusy THEN
				IF fbFileClose.bError THEN
					nErrorId := UDINT_TO_UINT(fbFileClose.nErrId);
					bError := TRUE;
					nStateA_LoadSaveDel := 99;				
				ELSE
					bConfigSaved := TRUE;
					fbSettings.M_WritePersData();
					nStateA_LoadSaveDel := 80;
				END_IF
				fbFileClose(hFile:= hFile, bExecute:= FALSE);
				bBusy := FALSE;
			END_IF
		ELSE
			bBusy := FALSE;
		END_IF
		IF NOT bBusy AND nStateA_LoadSaveDel = 99 THEN
			bError := TRUE;
		END_IF
	END_IF
ELSE
	nStateA_LoadSaveDel := 0;
	bError := FALSE;
END_IF
END_ACTION

ACTION A_Load:
IF bExecute THEN
	IF nStateA_LoadSaveDel = 0 THEN //File "Standard.cfg" zum Lesen öffnen
		bBusy := TRUE;
		hFile := 0;
		fbFileOpen(sPathName:= sConfigPath, nMode:= FOPEN_MODEREAD OR FOPEN_MODEBINARY, bExecute:= TRUE);
		IF NOT fbFileOpen.bBusy THEN
			IF fbFileOpen.bError THEN
				nErrorId := UDINT_TO_UINT(fbFileOpen.nErrId);
				nStateA_LoadSaveDel := 99;
			ELSE
				hFile := fbFileOpen.hFile;
				nStateA_LoadSaveDel := 1;
			END_IF
			fbFileOpen(bExecute:= FALSE);
		END_IF
	END_IF
	
	IF nStateA_LoadSaveDel = 1 THEN //Anzahl der zu lesenden Bytes für den ersten Datensatz lesen
		fbFileRead(hFile:= hFile, pReadBuff:= ADR(nBytesNextRead), cbReadLen:= SIZEOF(nBytesNextRead), bExecute:= TRUE);
		IF NOT fbFileRead.bBusy THEN
			IF fbFileRead.bError THEN
				nErrorId := UDINT_TO_UINT(fbFileRead.nErrId);
				nStateA_LoadSaveDel := 99;
			ELSE
				nStateA_LoadSaveDel := 2;
				MEMSET(ADR(stPropData),0,SIZEOF(stPropData));
			END_IF
			fbFileRead(bExecute:= FALSE);
		END_IF
	END_IF
	
	IF nStateA_LoadSaveDel = 2 THEN
		//solange Datensätze einlesen bis EOF kommt
		//es werden 2Bytes mehr gelesen (nBytes des nächsten Datensatzes
		fbFileRead(hFile:= hFile, pReadBuff:= ADR(stPropData), cbReadLen:= nBytesNextRead, bExecute:= TRUE);
		IF NOT fbFileRead.bBusy THEN
			IF fbFileRead.bError THEN
				nErrorId := UDINT_TO_UINT(fbFileRead.nErrId);
				nStateA_LoadSaveDel := 99;
			ELSE
				//nBytesNextRead für nächsen Datensatz ermitteln
				MEMCPY(ADR(nBytesNextRead),ADR(stPropData) + nBytesNextRead - 2, 2);
				IF fbObjectDirectory.M_CreateObject(-1, stPropData) > 0 THEN
					nStateA_LoadSaveDel := 99;
				END_IF
				IF nBytesNextRead = 0 OR fbFileRead.bEOF THEN
					nStateA_LoadSaveDel := 3;
				END_IF
			END_IF
			fbFileRead(bExecute:= FALSE);
			MEMSET(ADR(stPropData),0,SIZEOF(stPropData));
		END_IF
	END_IF
	
	IF nStateA_LoadSaveDel = 3 OR nStateA_LoadSaveDel = 99 THEN
		IF hFile > 0 THEN
			fbFileClose(hFile:= hFile, bExecute:= TRUE);
			IF NOT fbFileClose.bBusy THEN
				IF fbFileClose.bError THEN
					nErrorId := UDINT_TO_UINT(fbFileClose.nErrId);
					bError := TRUE;
					nStateA_LoadSaveDel := 99;				
				ELSE
					nStateA_LoadSaveDel := 80;
				END_IF
				fbFileClose(hFile:= hFile, bExecute:= FALSE);
				bBusy := FALSE;
			END_IF
		ELSE
			bBusy := FALSE;
		END_IF
		IF NOT bBusy AND nStateA_LoadSaveDel = 99 THEN
			bError := TRUE;
		END_IF
	END_IF
ELSE
	nStateA_LoadSaveDel := 0;
	bError := FALSE;
END_IF
END_ACTION

METHOD M_Deactivate
VAR_INPUT
END_VAR
bActivated := FALSE;
END_METHOD

PROPERTY P_bActivated : BOOL
GET
P_bActivated := bActivated;
END_GET
END_PROPERTY

PROPERTY P_bConfigSaved : BOOL
GET
P_bConfigSaved := bConfigSaved;
END_GET
END_PROPERTY

END_FUNCTION_BLOCK

// ---- Hardware/Settings/FB_Settings.TcPOU
FUNCTION_BLOCK FB_Settings

VAR
	bWritePersData	: BOOL;
	nStateA_WritePersData	: USINT := 80;
	tmrWritePersData		: TON;
	fbWritePersistentData	: WritePersistentData;
END_VAR

//Die persitenten Daten werden erst 100ms nach Anforderung geschrieben
//jede erneute Anforderung setzt diesen Timer zurück, so dass nicht bei
//schnellen hinteraeinanderfolgenden Anforderungen nicht ständig alle Daten
//neu geschrieben werden
IF bWritePersData THEN
	IF nStateA_WritePersData = 0 THEN	//Timer zurücksetzen
		tmrWritePersData(IN:= FALSE);
		bWritePersData := FALSE;
	ELSIF nStateA_WritePersData = 80 THEN
		nStateA_WritePersData := 0;
		bWritePersData := FALSE;
	END_IF
END_IF
	
IF nStateA_WritePersData = 0 THEN
	tmrWritePersData(IN:= TRUE, PT:=T#100MS);
	IF tmrWritePersData.Q THEN
		nStateA_WritePersData := 1;
	END_IF
ELSIF nStateA_WritePersData = 1 THEN
	fbWritePersistentData(PORT:= 851, START:= TRUE);
	IF NOT fbWritePersistentData.BUSY THEN
		IF fbWritePersistentData.ERR THEN
			nStateA_WritePersData := 99;
		ELSE
			nStateA_WritePersData := 80;
		END_IF
		tmrWritePersData(IN:= FALSE);
		fbWritePersistentData(START:= FALSE);
	END_IF
END_IF

METHOD M_ReadProp : ERRORID
VAR_INPUT
	stHardwareId : ST_HardwareId;
	ePropType 	: E_HardwarePropType;
END_VAR
VAR_OUTPUT
	nValue : DINT;
END_VAR
VAR
	pXYDrive : POINTER TO FB_XYDriveBase;
	pTMCM1140Stepper : POINTER TO FB_HwRefTMCM1140;
END_VAR
CASE stHardwareId.eGroup OF
	E_HardwareGrp.AxisX,E_HardwareGrp.AxisY:
		pXYDrive := fbXYDriveList.M_GetByHwId(stHardwareId);
		IF pXYDrive > 0 THEN
			M_ReadProp := pXYDrive^.M_GetProperty(eType:= ePropType, nValue=> nValue);
		ELSE
			M_ReadProp := E_ErrorIdCmd.ERRORID_InvalidHwItem;
		END_IF

	E_HardwareGrp.AxisZ:
		IF stHardwareId.nParentItem > 0 AND stHardwareId.nParentItem <= cMaxMzHeads THEN
			IF stHardwareId.nItem >= 1 AND stHardwareId.nItem <= 7 THEN
				CASE ePropType OF
					E_HardwarePropType.RefPos1:
						nValue := REAL_TO_DINT(aFbMultiZRef[stHardwareId.nParentItem].aFbZAxisRef[stHardwareId.nItem].P_rRefPos);
					E_HardwarePropType.HomePos:
						nValue := REAL_TO_DINT(aFbMultiZRef[stHardwareId.nParentItem].aFbZAxisRef[stHardwareId.nItem].P_rHomePos);
					E_HardwarePropType.AxisLength:
						nValue := REAL_TO_DINT(aFbMultiZRef[stHardwareId.nParentItem].aFbZAxisRef[stHardwareId.nItem].P_rAxisLength);
					E_HardwarePropType.SliderLength:
						nValue := REAL_TO_DINT(aFbMultiZRef[stHardwareId.nParentItem].aFbZAxisRef[stHardwareId.nItem].P_rSliderLength);
					E_HardwarePropType.InvertInitDir:
						nValue := BOOL_TO_DINT(aFbMultiZRef[stHardwareId.nParentItem].aFbZAxisRef[stHardwareId.nItem].P_bInvertInitDir);						
					E_HardwarePropType.MinPos:
						nValue := REAL_TO_DINT(aFbMultiZRef[stHardwareId.nParentItem].aFbZAxisRef[stHardwareId.nItem].P_rMinPos);
					E_HardwarePropType.MaxPos:
						nValue := REAL_TO_DINT(aFbMultiZRef[stHardwareId.nParentItem].aFbZAxisRef[stHardwareId.nItem].P_rMaxPos);
					E_HardwarePropType.MaxSpeed:
						nValue := REAL_TO_DINT(aFbMultiZRef[stHardwareId.nParentItem].aFbZAxisRef[stHardwareId.nItem].P_rMaxSpeed);
				ELSE
					M_ReadProp := E_ErrorIdCmd.ERRORID_InvalidHwProperty;					
				END_CASE
			ELSE
				M_ReadProp := E_ErrorIdCmd.ERRORID_InvalidHwItem;	
			END_IF
 		ELSE
			M_ReadProp := E_ErrorIdCmd.ERRORID_InvalidHwItem;
		END_IF	
	
	E_HardwareGrp.PneuChannel:
		IF stHardwareId.nItem >= 1 AND stHardwareId.nItem <= cNoOfPneuChannels THEN
			CASE ePropType OF
				E_HardwarePropType.MinPress:
					nValue:= aFbPneuChannel[stHardwareId.nItem].P_nMinPress;
				E_HardwarePropType.MaxPress:
					nValue:= aFbPneuChannel[stHardwareId.nItem].P_nMaxPress;
				E_HardwarePropType.MinPressCV:
					nValue:= aFbPneuChannel[stHardwareId.nItem].P_nMinPressCV;
				E_HardwarePropType.MinPressMV:
					nValue:= aFbPneuChannel[stHardwareId.nItem].P_nMinPressMV;
				E_HardwarePropType.MaxPressCV:
					nValue:= aFbPneuChannel[stHardwareId.nItem].P_nMaxPressCV;
				E_HardwarePropType.MaxPressMV:
					nValue:= aFbPneuChannel[stHardwareId.nItem].P_nMaxPressMV;
				E_HardwarePropType.FactorSetPress:
					nValue:= aFbPneuChannel[stHardwareId.nItem].P_nFactSetPress;
				E_HardwarePropType.FactorCurrentPress:
					nValue:= aFbPneuChannel[stHardwareId.nItem].P_nFactCurrPress;
				E_HardwarePropType.OffsetSetPress:
					nValue:= aFbPneuChannel[stHardwareId.nItem].P_nOffsetSetPress;
				E_HardwarePropType.OffseCurrentPress:
					nValue:= aFbPneuChannel[stHardwareId.nItem].P_nOffsetCurrPress;				
			ELSE
				M_ReadProp := E_ErrorIdCmd.ERRORID_InvalidHwProperty;
			END_CASE			
		ELSE
			M_ReadProp := E_ErrorIdCmd.ERRORID_InvalidHwItem;
		END_IF
	E_HardwareGrp.StopButton:
		IF stHardwareId.nItem = 1 THEN
			IF ePropType = E_HardwarePropType.Disabled THEN
				nValue := BOOL_TO_DINT(fbStopButton.P_bDisabled);
			ELSE
				M_ReadProp := E_ErrorIdCmd.ERRORID_InvalidHwProperty;
			END_IF
		ELSE
			M_ReadProp := E_ErrorIdCmd.ERRORID_InvalidHwItem;
		END_IF
	E_HardwareGrp.HighVoltSupply:
		{IF defined(variable:fbHighVoltSupplyRef)}
		IF stHardwareId.nItem = 1 THEN
			CASE ePropType OF
				E_HardwarePropType.MinVoltage:
					nValue := fbHighVoltSupplyRef.P_nMinVoltage;
				E_HardwarePropType.MaxVoltage:
					nValue := fbHighVoltSupplyRef.P_nMaxVoltage;
				E_HardwarePropType.MinVoltageCV:
					nValue := fbHighVoltSupplyRef.P_nMinVoltageCV;
				E_HardwarePropType.MaxVoltageCV:
					nValue := fbHighVoltSupplyRef.P_nMaxVoltageCV;
				E_HardwarePropType.MinVoltageMV:
					nValue := fbHighVoltSupplyRef.P_nMinVoltageMV;
				E_HardwarePropType.MaxVoltageMV:
					nValue := fbHighVoltSupplyRef.P_nMaxVoltageMV;
				E_HardwarePropType.MinCurrent:
					nValue := fbHighVoltSupplyRef.P_nMinCurrent;
				E_HardwarePropType.MaxCurrent:
					nValue := fbHighVoltSupplyRef.P_nMaxCurrent;
				E_HardwarePropType.MinCurrentCV:
					nValue := fbHighVoltSupplyRef.P_nMinCurrentCV;
				E_HardwarePropType.MaxCurrentCV:
					nValue := fbHighVoltSupplyRef.P_nMaxCurrentCV;
				E_HardwarePropType.MinCurrentMV:
					nValue := fbHighVoltSupplyRef.P_nMinCurrentMV;
				E_HardwarePropType.MaxCurrentMV:
					nValue := fbHighVoltSupplyRef.P_nMaxCurrentMV;
				E_HardwarePropType.Legacy:
					nValue := BOOL_TO_DINT(fbHighVoltSupplyRef.P_bLegacy);
			ELSE
				M_ReadProp := E_ErrorIdCmd.ERRORID_InvalidHwProperty;
			END_CASE
		ELSE
			M_ReadProp := E_ErrorIdCmd.ERRORID_InvalidHwItem;
		END_IF
		{ELSE}
		M_ReadProp := E_ErrorIdCmd.ERRORID_InvalidHwItem;
		{END_IF}
	E_HardwareGrp.NanotecPD:
		{IF defined(variable:fbHwRefTrayTransSlider)}
		IF stHardwareId.nItem = 1 THEN
			CASE ePropType OF
				E_HardwarePropType.DistPerMotorRev:	
					nValue := fbHwRefTrayTransSlider.P_nDistPerMotorRev;
				E_HardwarePropType.RefPos1:
					nValue := fbHwRefTrayTransSlider.P_nRefPos;
				E_HardwarePropType.HomePos:
					nValue := fbHwRefTrayTransSlider.P_nHomePos;
				E_HardwarePropType.SlowHomingSpeed:
					nValue := fbHwRefTrayTransSlider.P_nSlowHomingSpeed;
				E_HardwarePropType.FastHomingSpeed:
					nValue := fbHwRefTrayTransSlider.P_nFastHomingSpeed;
				E_HardwarePropType.InvertInitDir:
					nValue := BOOL_TO_DINT(fbHwRefTrayTransSlider.P_bInvertInitDir);
				E_HardwarePropType.MinPos:
					nValue := fbHwRefTrayTransSlider.P_nMinPos;
				E_HardwarePropType.MaxPos:
					nValue := fbHwRefTrayTransSlider.P_nMaxPos;
				E_HardwarePropType.MaxSpeed:
					nValue := fbHwRefTrayTransSlider.P_nMaxSpeed;
			ELSE
				M_ReadProp := E_ErrorIdCmd.ERRORID_InvalidHwProperty;
			END_CASE
		ELSE
			M_ReadProp := E_ErrorIdCmd.ERRORID_InvalidHwItem;	
		END_IF
		{ELSE}
		M_ReadProp := E_ErrorIdCmd.ERRORID_InvalidHwItem;
		{END_IF}
	E_HardwareGrp.TMCM1140Stepper_Gen2:
		pTMCM1140Stepper := fbCANOpenHwModuleList.M_GetByHwId(stHardwareId);
		IF pTMCM1140Stepper > 0 THEN
			CASE ePropType OF
					E_HardwarePropType.DistPerMotorRev:	
						nValue := pTMCM1140Stepper^.P_nDistPerMotorRev;
					E_HardwarePropType.RefPos1:
						nValue := pTMCM1140Stepper^.P_nRefPos;
					E_HardwarePropType.HomePos:
						nValue := pTMCM1140Stepper^.P_nHomePos;
					E_HardwarePropType.SlowHomingSpeed:
						nValue := pTMCM1140Stepper^.P_nSlowHomingSpeed;
					E_HardwarePropType.FastHomingSpeed:
						nValue := pTMCM1140Stepper^.P_nFastHomingSpeed;
					(*E_HardwarePropType.InvertInitDir:
						fbHwRefTrayTransSlider.P_bInvertInitDir := DINT_TO_BOOL(nValue);*)
					E_HardwarePropType.MinPos:
						nValue := pTMCM1140Stepper^.P_nMinPos;
					E_HardwarePropType.MaxPos:
						nValue := pTMCM1140Stepper^.P_nMaxPos;
					E_HardwarePropType.MaxSpeed:
						nValue := pTMCM1140Stepper^.P_nMaxSpeed;
					E_HardwarePropType.MaxCurrent:
						nValue := pTMCM1140Stepper^.P_nMaxCurrent;
					E_HardwarePropType.HoldCurrent:
						nValue := pTMCM1140Stepper^.P_nHoldCurrent;
			END_CASE		
		ELSE
			M_ReadProp := E_ErrorIdCmd.ERRORID_InvalidHwItem;
		END_IF
	E_HardwareGrp.EL70xx:
		IF stHardwareId.nItem = 1 THEN
			{IF defined(variable:fbHwRefSpinDrive)}
			CASE ePropType OF
				E_HardwarePropType.DistPerMotorRev:	
					nValue := fbHwRefSpinDrive.P_nDistPerMotorRev;
				E_HardwarePropType.RefPos1:
					nValue := fbHwRefSpinDrive.P_nRefPos;
				E_HardwarePropType.InvertInitDir:
					nValue := BOOL_TO_DINT(fbHwRefSpinDrive.P_bInvertInitDir);
				E_HardwarePropType.MinPos:
					nValue := fbHwRefSpinDrive.P_nMinPos;
				E_HardwarePropType.MaxPos:
					nValue := fbHwRefSpinDrive.P_nMaxPos;
				E_HardwarePropType.MaxSpeed:
					nValue := fbHwRefSpinDrive.P_nMaxSpeed;
			ELSE
				M_ReadProp := E_ErrorIdCmd.ERRORID_InvalidHwProperty;
			END_CASE
			{ELSE}
			M_ReadProp := E_ErrorIdCmd.ERRORID_InvalidHwItem;
			{END_IF}			
		ELSIF stHardwareId.nItem = 2 THEN
			{IF defined(variable:fbHwRefLiftDrive)}
			CASE ePropType OF
				E_HardwarePropType.DistPerMotorRev:	
					nValue := fbHwRefLiftDrive.P_nDistPerMotorRev;
				E_HardwarePropType.RefPos1:
					nValue := fbHwRefLiftDrive.P_nRefPos;
				E_HardwarePropType.InvertInitDir:
					nValue := BOOL_TO_DINT(fbHwRefLiftDrive.P_bInvertInitDir);
				E_HardwarePropType.MinPos:
					nValue := fbHwRefLiftDrive.P_nMinPos;
				E_HardwarePropType.MaxPos:
					nValue := fbHwRefLiftDrive.P_nMaxPos;
				E_HardwarePropType.MaxSpeed:
					nValue := fbHwRefLiftDrive.P_nMaxSpeed;
			ELSE
				M_ReadProp := E_ErrorIdCmd.ERRORID_InvalidHwProperty;
			END_CASE
			{ELSE}
			M_ReadProp := E_ErrorIdCmd.ERRORID_InvalidHwItem;
			{END_IF}			
		ELSIF stHardwareId.nItem = 3 THEN
			{IF defined(variable:fbHwRefTrayStop)}
			CASE ePropType OF
				E_HardwarePropType.DistPerMotorRev:	
					nValue := fbHwRefTrayStop.P_nDistPerMotorRev;
				E_HardwarePropType.RefPos1:
					nValue := fbHwRefTrayStop.P_nRefPos;
				E_HardwarePropType.InvertInitDir:
					nValue := BOOL_TO_DINT(fbHwRefTrayStop.P_bInvertInitDir);
				E_HardwarePropType.MinPos:
					nValue := fbHwRefTrayStop.P_nMinPos;
				E_HardwarePropType.MaxPos:
					nValue := fbHwRefTrayStop.P_nMaxPos;
				E_HardwarePropType.MaxSpeed:
					nValue := fbHwRefTrayStop.P_nMaxSpeed;
			ELSE
				M_ReadProp := E_ErrorIdCmd.ERRORID_InvalidHwProperty;
			END_CASE
			{ELSE}
			M_ReadProp := E_ErrorIdCmd.ERRORID_InvalidHwItem;
			{END_IF}			
		ELSE
			M_ReadProp := E_ErrorIdCmd.ERRORID_InvalidHwItem;
		END_IF	
ELSE
	M_ReadProp := E_ErrorIdCmd.ERRORID_InvalidHwGroup;
END_CASE
END_METHOD

METHOD M_WritePersData
VAR_INPUT
END_VAR
bWritePersData := TRUE;
END_METHOD

METHOD M_WriteProp : ERRORID
VAR_INPUT
	stHardwareId : ST_HardwareId;
	ePropType : E_HardwarePropType;	
	nValue : DINT;
END_VAR
VAR
	pXYDrive : POINTER TO FB_XYDriveBase;
	pTMCM1140Stepper : POINTER TO FB_HwRefTMCM1140;
END_VAR
CASE stHardwareId.eGroup OF
	E_HardwareGrp.AxisX, E_HardwareGrp.AxisY:
		pXYDrive := fbXYDriveList.M_GetByHwId(stHardwareId);
		IF pXYDrive > 0 THEN
			M_WriteProp := pXYDrive^.M_SetProperty(ePropType, nValue);
		ELSE
			M_WriteProp := E_ErrorIdCmd.ERRORID_InvalidHwItem;
		END_IF		
		
	E_HardwareGrp.AxisZ:
		IF stHardwareId.nParentItem > 0 AND stHardwareId.nParentItem <= cMaxMzHeads THEN
			IF stHardwareId.nItem >= 1 AND stHardwareId.nItem <= 7 THEN
				CASE ePropType OF
					E_HardwarePropType.RefPos1:
						aFbMultiZRef[stHardwareId.nParentItem].aFbZAxisRef[stHardwareId.nItem].P_rRefPos := DINT_TO_REAL(nValue);
					E_HardwarePropType.HomePos:
						aFbMultiZRef[stHardwareId.nParentItem].aFbZAxisRef[stHardwareId.nItem].P_rHomePos := DINT_TO_REAL(nValue);
					E_HardwarePropType.AxisLength:
						aFbMultiZRef[stHardwareId.nParentItem].aFbZAxisRef[stHardwareId.nItem].P_rAxisLength := DINT_TO_REAL(nValue);
					E_HardwarePropType.SliderLength:
						aFbMultiZRef[stHardwareId.nParentItem].aFbZAxisRef[stHardwareId.nItem].P_rSliderLength := DINT_TO_REAL(nValue);
					E_HardwarePropType.InvertInitDir:
						aFbMultiZRef[stHardwareId.nParentItem].aFbZAxisRef[stHardwareId.nItem].P_bInvertInitDir := DINT_TO_BOOL(nValue);
					E_HardwarePropType.MinPos:
						aFbMultiZRef[stHardwareId.nParentItem].aFbZAxisRef[stHardwareId.nItem].P_rMinPos := DINT_TO_REAL(nValue);
					E_HardwarePropType.MaxPos:
						aFbMultiZRef[stHardwareId.nParentItem].aFbZAxisRef[stHardwareId.nItem].P_rMaxPos := DINT_TO_REAL(nValue);
					E_HardwarePropType.MaxSpeed:
					aFbMultiZRef[stHardwareId.nParentItem].aFbZAxisRef[stHardwareId.nItem].P_rMaxSpeed := DINT_TO_REAL(nValue);
				ELSE
					M_WriteProp := E_ErrorIdCmd.ERRORID_InvalidHwProperty;					
				END_CASE
			ELSE
				M_WriteProp := E_ErrorIdCmd.ERRORID_InvalidHwItem;	
			END_IF
 		ELSE
			M_WriteProp := E_ErrorIdCmd.ERRORID_InvalidHwItem;
		END_IF
		
	E_HardwareGrp.PneuChannel:
		IF stHardwareId.nItem >= 1 AND stHardwareId.nItem <= cNoOfPneuChannels THEN
			CASE ePropType OF
				E_HardwarePropType.MinPress:
					aFbPneuChannel[stHardwareId.nItem].P_nMinPress := nValue;
				E_HardwarePropType.MaxPress:
					aFbPneuChannel[stHardwareId.nItem].P_nMaxPress := nValue;
				E_HardwarePropType.MinPressCV:
					aFbPneuChannel[stHardwareId.nItem].P_nMinPressCV := nValue;
				E_HardwarePropType.MinPressMV:
					aFbPneuChannel[stHardwareId.nItem].P_nMinPressMV := nValue;
				E_HardwarePropType.MaxPressCV:
					aFbPneuChannel[stHardwareId.nItem].P_nMaxPressCV := nValue;
				E_HardwarePropType.MaxPressMV:
					aFbPneuChannel[stHardwareId.nItem].P_nMaxPressMV := nValue;
				E_HardwarePropType.FactorSetPress:
						aFbPneuChannel[stHardwareId.nItem].P_nFactSetPress := nValue;
				E_HardwarePropType.FactorCurrentPress:
					aFbPneuChannel[stHardwareId.nItem].P_nFactCurrPress := nValue;
				E_HardwarePropType.OffsetSetPress:
					aFbPneuChannel[stHardwareId.nItem].P_nOffsetSetPress := nValue;
				E_HardwarePropType.OffseCurrentPress:
					aFbPneuChannel[stHardwareId.nItem].P_nOffsetCurrPress := nValue;
			ELSE
				M_WriteProp := E_ErrorIdCmd.ERRORID_InvalidHwProperty;
			END_CASE
		ELSE
			M_WriteProp := E_ErrorIdCmd.ERRORID_InvalidHwItem;			
		END_IF
	E_HardwareGrp.StopButton:
		IF stHardwareId.nItem = 1 THEN
			IF ePropType = E_HardwarePropType.Disabled THEN
				fbStopButton.P_bDisabled := DINT_TO_BOOL(nValue);
			ELSE
				M_WriteProp := E_ErrorIdCmd.ERRORID_InvalidHwProperty;
			END_IF
		ELSE
			M_WriteProp := E_ErrorIdCmd.ERRORID_InvalidHwItem;
		END_IF
	E_HardwareGrp.HighVoltSupply:
		{IF defined(variable:fbHighVoltSupplyRef)}
		IF stHardwareId.nItem = 1 THEN
			CASE ePropType OF
				E_HardwarePropType.MinVoltage:
					fbHighVoltSupplyRef.P_nMinVoltage := nValue;
				E_HardwarePropType.MaxVoltage:
					fbHighVoltSupplyRef.P_nMaxVoltage := nValue;
				E_HardwarePropType.MinVoltageCV:
					fbHighVoltSupplyRef.P_nMinVoltageCV := nValue;
				E_HardwarePropType.MaxVoltageCV:
					fbHighVoltSupplyRef.P_nMaxVoltageCV := nValue;
				E_HardwarePropType.MinVoltageMV:
					fbHighVoltSupplyRef.P_nMinVoltageMV := nValue;
				E_HardwarePropType.MaxVoltageMV:
					fbHighVoltSupplyRef.P_nMaxVoltageMV := nValue;
				E_HardwarePropType.MinCurrent:
					fbHighVoltSupplyRef.P_nMinCurrent := nValue;
				E_HardwarePropType.MaxCurrent:
					fbHighVoltSupplyRef.P_nMaxCurrent := nValue;
				E_HardwarePropType.MinCurrentCV:
					fbHighVoltSupplyRef.P_nMinCurrentCV := nValue;
				E_HardwarePropType.MaxCurrentCV:
					fbHighVoltSupplyRef.P_nMaxCurrentCV := nValue;
				E_HardwarePropType.MinCurrentMV:
					fbHighVoltSupplyRef.P_nMinCurrentMV := nValue;
				E_HardwarePropType.MaxCurrentMV:
					fbHighVoltSupplyRef.P_nMaxCurrentMV := nValue;
				E_HardwarePropType.Legacy:
					fbHighVoltSupplyRef.P_bLegacy := DINT_TO_BOOL(nValue);
			ELSE
				M_WriteProp := E_ErrorIdCmd.ERRORID_InvalidHwProperty;
			END_CASE
		ELSE
			M_WriteProp := E_ErrorIdCmd.ERRORID_InvalidHwItem;
		END_IF
		{ELSE}
		M_WriteProp := E_ErrorIdCmd.ERRORID_InvalidHwItem;
		{END_IF}
	E_HardwareGrp.NanotecPD:
		{IF defined(variable:fbHwRefTrayTransSlider)}
		IF stHardwareId.nItem = 1 THEN
			CASE ePropType OF
				E_HardwarePropType.DistPerMotorRev:	
					fbHwRefTrayTransSlider.P_nDistPerMotorRev := nValue;
				E_HardwarePropType.RefPos1:
					fbHwRefTrayTransSlider.P_nRefPos := nValue;
				E_HardwarePropType.HomePos:
					fbHwRefTrayTransSlider.P_nHomePos := nValue;
				E_HardwarePropType.SlowHomingSpeed:
					fbHwRefTrayTransSlider.P_nSlowHomingSpeed := nValue;
				E_HardwarePropType.FastHomingSpeed:
					fbHwRefTrayTransSlider.P_nFastHomingSpeed := nValue;
				E_HardwarePropType.InvertInitDir:
					fbHwRefTrayTransSlider.P_bInvertInitDir := DINT_TO_BOOL(nValue);
				E_HardwarePropType.MinPos:
					fbHwRefTrayTransSlider.P_nMinPos := nValue;
				E_HardwarePropType.MaxPos:
					fbHwRefTrayTransSlider.P_nMaxPos := nValue;
				E_HardwarePropType.MaxSpeed:
					fbHwRefTrayTransSlider.P_nMaxSpeed := nValue;
			ELSE
				M_WriteProp := E_ErrorIdCmd.ERRORID_InvalidHwProperty;
			END_CASE
		ELSE
			M_WriteProp := E_ErrorIdCmd.ERRORID_InvalidHwItem;
		END_IF
		{ELSE}
		M_WriteProp := E_ErrorIdCmd.ERRORID_InvalidHwItem;
		{END_IF}
	E_HardwareGrp.TMCM1140Stepper_Gen2:
		pTMCM1140Stepper := fbCANOpenHwModuleList.M_GetByHwId(stHardwareId);
		IF pTMCM1140Stepper > 0 THEN
			CASE ePropType OF
					E_HardwarePropType.DistPerMotorRev:	
						pTMCM1140Stepper^.P_nDistPerMotorRev := nValue;
					E_HardwarePropType.RefPos1:
						pTMCM1140Stepper^.P_nRefPos := nValue;
					E_HardwarePropType.HomePos:
						pTMCM1140Stepper^.P_nHomePos := nValue;
					E_HardwarePropType.SlowHomingSpeed:
						pTMCM1140Stepper^.P_nSlowHomingSpeed := nValue;
					E_HardwarePropType.FastHomingSpeed:
						pTMCM1140Stepper^.P_nFastHomingSpeed := nValue;
					(*E_HardwarePropType.InvertInitDir:
						fbHwRefTrayTransSlider.P_bInvertInitDir := DINT_TO_BOOL(nValue);*)
					E_HardwarePropType.MinPos:
						pTMCM1140Stepper^.P_nMinPos := nValue;
					E_HardwarePropType.MaxPos:
						pTMCM1140Stepper^.P_nMaxPos := nValue;
					E_HardwarePropType.MaxSpeed:
						pTMCM1140Stepper^.P_nMaxSpeed := nValue;
					E_HardwarePropType.MaxCurrent:
						pTMCM1140Stepper^.P_nMaxCurrent := DINT_TO_UINT(nValue);
					E_HardwarePropType.HoldCurrent:
						pTMCM1140Stepper^.P_nHoldCurrent := DINT_TO_UINT(nValue);
			END_CASE		
		ELSE
			M_WriteProp := E_ErrorIdCmd.ERRORID_InvalidHwItem;
		END_IF
	E_HardwareGrp.EL70xx:
		IF stHardwareId.nItem = 1 THEN
			{IF defined(variable:fbHwRefSpinDrive)}
			CASE ePropType OF
				E_HardwarePropType.DistPerMotorRev:	
					fbHwRefSpinDrive.P_nDistPerMotorRev := nValue;
				E_HardwarePropType.RefPos1:
					fbHwRefSpinDrive.P_nRefPos := nValue;
				E_HardwarePropType.InvertInitDir:
					fbHwRefSpinDrive.P_bInvertInitDir := DINT_TO_BOOL(nValue);
				E_HardwarePropType.MinPos:
					fbHwRefSpinDrive.P_nMinPos := nValue;
				E_HardwarePropType.MaxPos:
					fbHwRefSpinDrive.P_nMaxPos := nValue;
				E_HardwarePropType.MaxSpeed:
					fbHwRefSpinDrive.P_nMaxSpeed := nValue;
			ELSE
				M_WriteProp := E_ErrorIdCmd.ERRORID_InvalidHwProperty;
			END_CASE
			{ELSE}
			M_WriteProp := E_ErrorIdCmd.ERRORID_InvalidHwItem;
			{END_IF}			
		ELSIF stHardwareId.nItem = 2 THEN
			{IF defined(variable:fbHwRefLiftDrive)}
			CASE ePropType OF
				E_HardwarePropType.DistPerMotorRev:	
					fbHwRefLiftDrive.P_nDistPerMotorRev := nValue;
				E_HardwarePropType.RefPos1:
					fbHwRefLiftDrive.P_nRefPos := nValue;
				E_HardwarePropType.InvertInitDir:
					fbHwRefLiftDrive.P_bInvertInitDir := DINT_TO_BOOL(nValue);
				E_HardwarePropType.MinPos:
					fbHwRefLiftDrive.P_nMinPos := nValue;
				E_HardwarePropType.MaxPos:
					fbHwRefLiftDrive.P_nMaxPos := nValue;
				E_HardwarePropType.MaxSpeed:
					fbHwRefLiftDrive.P_nMaxSpeed := nValue;
			ELSE
				M_WriteProp := E_ErrorIdCmd.ERRORID_InvalidHwProperty;
			END_CASE
			{ELSE}
			M_WriteProp := E_ErrorIdCmd.ERRORID_InvalidHwItem;
			{END_IF}			
		ELSIF stHardwareId.nItem = 3 THEN
			{IF defined(variable:fbHwRefTrayStop)}
			CASE ePropType OF
				E_HardwarePropType.DistPerMotorRev:	
					fbHwRefTrayStop.P_nDistPerMotorRev := nValue;
				E_HardwarePropType.RefPos1:
					fbHwRefTrayStop.P_nRefPos := nValue;
				E_HardwarePropType.InvertInitDir:
					fbHwRefTrayStop.P_bInvertInitDir := DINT_TO_BOOL(nValue);
				E_HardwarePropType.MinPos:
					fbHwRefTrayStop.P_nMinPos := nValue;
				E_HardwarePropType.MaxPos:
					fbHwRefTrayStop.P_nMaxPos := nValue;
				E_HardwarePropType.MaxSpeed:
					fbHwRefTrayStop.P_nMaxSpeed := nValue;
			ELSE
				M_WriteProp := E_ErrorIdCmd.ERRORID_InvalidHwProperty;
			END_CASE
			{ELSE}
			M_WriteProp := E_ErrorIdCmd.ERRORID_InvalidHwItem;
			{END_IF}			
		ELSE
			M_WriteProp := E_ErrorIdCmd.ERRORID_InvalidHwItem;
		END_IF
ELSE
	M_WriteProp := E_ErrorIdCmd.ERRORID_InvalidHwGroup;		
END_CASE
END_METHOD

END_FUNCTION_BLOCK

// ---- Hardware/FB_HwModuleList.TcPOU
FUNCTION_BLOCK FB_HwModuleList
VAR_INPUT
END_VAR
VAR_OUTPUT
END_VAR
VAR
	pHead	: POINTER TO ST_Pointer;
	pTail	: POINTER TO ST_Pointer;
	pCurrent: POINTER TO ST_Pointer;
	nCount	: UINT;	
END_VAR

METHOD FB_exit : BOOL
VAR_INPUT
	bInCopyCode : BOOL; // if TRUE, the exit method is called for exiting an instance that is copied afterwards (online change).
END_VAR

VAR
	pPointer : POINTER TO ST_Pointer;
END_VAR
(*pPointer := pHead;
WHILE pPointer > 0 DO
	__DELETE(pPointer);
	pPointer := pPointer^.pNext;
END_WHILE*)
END_METHOD

METHOD M_Add
VAR_INPUT
	pModule : POINTER TO FB_HwModule;
END_VAR

VAR
	pNew : POINTER TO ST_Pointer;
END_VAR
pNew := pHead;
WHILE pNew > 0 DO
	IF pNew^.pContent = pModule THEN
		RETURN;
	END_IF
	pNew := pNew^.pNext;
END_WHILE

pNew := __NEW(ST_Pointer);
MEMSET(pNew,0,SIZEOF(ST_Pointer));
pNew^.pContent := pModule;
IF pHead = 0 THEN
	pHead := pTail := pNew;
ELSE
	pNew^.pPrev := pTail; 
	pTail^.pNext := pNew;
	pTail := pNew;
END_IF
nCount := nCount + 1;
END_METHOD

METHOD M_CountByGroup : UINT
VAR_INPUT
	eGroup : E_HardwareGrp;
END_VAR


VAR
	pPointer : POINTER TO ST_Pointer;
	pModule : POINTER TO FB_HwModule;
	stHwIdTemp : ST_HardwareId;
	nCount : UINT;
END_VAR
pPointer := pHead;
WHILE pPointer > 0 DO
	pModule := pPointer^.pContent;
	stHwIdTemp := pModule^.P_stHardwareId;
	IF eGroup = stHwIdTemp.eGroup THEN
		nCount := nCount + 1;
	END_IF
	pPointer := pPointer^.pNext;
END_WHILE
M_CountByGroup := nCount;
END_METHOD

METHOD M_Get : POINTER TO FB_HwModule
VAR_INPUT
END_VAR

VAR
	pModule : POINTER TO FB_HwModule;
END_VAR
IF pCurrent > 0 THEN
	pModule := pCurrent^.pContent;
	IF pModule > 0 THEN
		M_Get := pModule;
	END_IF
	pCurrent := pCurrent^.pNext;
END_IF
END_METHOD

METHOD M_GetByHwId : POINTER TO FB_HwModule
VAR_INPUT
	stHardwareId : ST_HardwareId;
END_VAR

VAR
	pPointer : POINTER TO ST_Pointer;
	pModule : POINTER TO FB_HwModule;
	stHwIdTemp : ST_HardwareId;
END_VAR
pPointer := pHead;
WHILE pPointer > 0 DO
	pModule := pPointer^.pContent;
	stHwIdTemp := pModule^.P_stHardwareId;
	//Strukturen können nicht direkt miteinander verglichen werden
	//IF stHwIdTemp = stHardwareId THEN
	IF MEMCMP(ADR(stHwIdTemp), ADR(stHardwareId), SIZEOF(ST_HardwareId)) = 0 THEN
		M_GetByHwId := pModule;
		RETURN;
	END_IF
	pPointer := pPointer^.pNext;
END_WHILE
END_METHOD

METHOD M_Reset
VAR_INPUT
END_VAR

VAR
	pDelete : POINTER TO ST_Pointer;
	pNext	: POINTER TO ST_Pointer;
END_VAR
pDelete := pHead;
WHILE  pDelete > 0 DO
	pNext := pDelete^.pNext;
	__DELETE(pDelete);
	pDelete := pNext;
END_WHILE
pHead := 0;
pTail := 0;
pCurrent := 0;
nCount := 0;
END_METHOD

METHOD M_SetCurrentToHead : BOOL
VAR_INPUT
END_VAR
pCurrent := pHead;
END_METHOD

END_FUNCTION_BLOCK

// ---- Hardware/BottleRack/FB_HwRefBottleRack.TcPOU
FUNCTION_BLOCK FB_HwRefBottleRack EXTENDS FB_CanNodeBase
VAR_INPUT
END_VAR
VAR_OUTPUT
	
END_VAR
VAR
	
END_VAR

IF bNodeEnabled THEN
	SUPER^();	
END_IF

ACTION A_ResetApp:
IF nStateA_ResetApp = 0 THEN
	fbSdoWrite(sADSNetID:= stAdsAdress.sNetId, nPortNr:= stAdsAdress.nPort,
				nIndex := cUpdateRequest.nIndex, nSubIndex := 0, nDataLength := 1, nData:= 1, bExecute:= TRUE);
	IF NOT fbSdoWrite.bBusy THEN
		IF fbSdoWrite.bError THEN
			nErrorId := fbSdoWrite.nAdsErrorId;
			nErrorId2 := fbSdoWrite.nSdoErrorId;
			nStateA_ResetApp := 99;  //Error
		ELSE
			nStateA_ResetApp := 80;
		END_IF
		fbSdoWrite(bExecute:= FALSE);
	END_IF
END_IF
END_ACTION

END_FUNCTION_BLOCK

// ---- Hardware/IOExpander/FB_HwRefIOExpander.TcPOU
FUNCTION_BLOCK FB_HwRefIOExpander EXTENDS FB_CanNodeBase
VAR_INPUT
END_VAR
VAR_OUTPUT
END_VAR
VAR
	//PDOs
	aInput			AT %I* : ARRAY[1..6] OF UINT;
	aOutput			AT %Q* : ARRAY[1..6] OF UINT;
	
	//Parameter für PulseTrain-Ausgänge
	//aPeriod 		AT %Q* : ARRAY[4..6] OF UINT;
	//aPulse 			AT %Q* : ARRAY[4..6] OF UINT;
	//aPulseNumber 	AT %Q* : ARRAY[4..6] OF UINT;
	aPulseTrainChannel : ARRAY[1..3] OF ST_PulseTrainChannel;

		
END_VAR

IF bNodeEnabled THEN
	SUPER^();
END_IF

ACTION A_ResetApp:
IF nStateA_ResetApp = 0 THEN
	fbSdoWrite(sADSNetID:= stAdsAdress.sNetId, nPortNr:= stAdsAdress.nPort,
				nIndex := cUpdateRequest.nIndex, nSubIndex := 0, nDataLength := 1, nData:= 1, bExecute:= TRUE);
	IF NOT fbSdoWrite.bBusy THEN
		IF fbSdoWrite.bError THEN
			nErrorId := fbSdoWrite.nAdsErrorId;
			nErrorId2 := fbSdoWrite.nSdoErrorId;
			nStateA_ResetApp := 99;  //Error
		ELSE
			nStateA_ResetApp := 80;
		END_IF
		fbSdoWrite(bExecute:= FALSE);
	END_IF
END_IF
END_ACTION

METHOD M_GetPulseTrainChannel : POINTER TO ST_PulseTrainChannel
VAR_INPUT
	nChannel : USINT;
END_VAR
IF nChannel >= 1 AND nChannel <= 3 THEN
	M_GetPulseTrainChannel := ADR(aPulseTrainChannel[nChannel]);
END_IF
END_METHOD

END_FUNCTION_BLOCK

// ---- Hardware/EL70xxDrive/FB_HwRefEL70xxDriveExtEncoder.TcPOU
FUNCTION_BLOCK FB_HwRefEL70xxDriveExtEncoder EXTENDS FB_HwRefEL70xxDrive
VAR_INPUT
END_VAR
VAR_OUTPUT
	nExtEncoderValue	AT %I* : UDINT;
	bExtEncoderError	AT %I* : BOOL;	
END_VAR
VAR
	rPositionOffset		: REAL;	//Bei absolutem Encoder der Wert, an dem das Drive an Position "0" steht
								//wird über RefPos errechnet
	rActualPosition 	: REAL; //das ist die tatsächliche Position berechnet aus dem aktuellen Encoderwert.
	//nSetCounterValue	AT %Q* : UDINT; //wäre nur für relative Encoder interessant ?
	//bSetCounter		AT %Q* : BOOL;	//dito
	//bSetCounterDone	AT %I* : BOOL;	//dito
END_VAR

SUPER^();

ACTION A_CalcActPosition:
IF eEncoderType = E_EL70xx_EncoderType.ExternSingleturnAbs THEN
	rPositionOffset := 360.0 * DINT_TO_REAL(nRefPos) / UDINT_TO_REAL(nEncoderIncrements);
	IF nExtEncoderValue < DINT_TO_UDINT(nRefPos) THEN
		rActualPosition := (360.0 - rPositionOffset + 360.0 * UDINT_TO_REAL(nExtEncoderValue) / UDINT_TO_REAL(nEncoderIncrements));
	ELSE
		rActualPosition := 360.0 * UDINT_TO_REAL(nExtEncoderValue) / UDINT_TO_REAL(nEncoderIncrements)- rPositionOffset;
	END_IF	
END_IF
nActualPosition := REAL_TO_DINT(rActualPosition * 1000.0);	//Integer als milliGrad oder µm
END_ACTION

ACTION A_Prepare:
//In dieser Klasse dürfen nur externe Encoder definiert sein.
IF eEncoderType <> E_EL70xx_EncoderType.ExternSingleturnAbs THEN
	nStateA_Prepare := 99;
END_IF
SUPER^.A_Prepare();
END_ACTION

METHOD FB_init : BOOL
VAR_INPUT
	bInitRetains 	: BOOL; 	// if TRUE, the retain variables are initialized (warm start / cold start)
	bInCopyCode  	: BOOL;  	// if TRUE, the instance afterwards gets moved into the copy code (online change)
	nBoxAddress		: UINT;
	eHomingMode		: E_EL70xx_StartType;
	eEncoderType	: E_EL70xx_EncoderType;
	nEnoderIncrements : UDINT;	
END_VAR

VAR
END_VAR
THIS^.eEncoderType := eEncoderType;
THIS^.nEncoderIncrements := nEnoderIncrements;
END_METHOD

METHOD M_GetPosDiff : DINT
VAR_INPUT
	nSetPosition : DINT;
END_VAR
IF nActualPosition > 359000 THEN //dann steht die aktuelle Position kurz über der Nullmarke
   M_GetPosDiff := nSetPosition - (P_nActualPosition - 360000);
ELSE
	M_GetPosDiff := nSetPosition - P_nActualPosition;
END_IF
END_METHOD

METHOD M_SetTargetPos : BOOL
VAR_INPUT
	nValue : DINT; //Reale Einheit
END_VAR
IF (nValue >= nMinPos) AND (nValue <= nMaxPos) THEN
	//Wenn sich Position zwischen 355° und 360° befindet, dann muss die Drehrichtung geändert werden
	IF nActualPosition > 355000 THEN
		POS_Control.TargetPosition := REAL_TO_DINT(DINT_TO_REAL(nValue - nActualPosition + 360000) *  rTranslationFactorPosition);
	ELSE
		POS_Control.TargetPosition := REAL_TO_DINT(DINT_TO_REAL(nValue - nActualPosition) * rTranslationFactorPosition);	
	END_IF
	POS_Control.StartType := E_EL70xx_StartType.Relative;
	M_SetTargetPos := TRUE;
END_IF
END_METHOD

END_FUNCTION_BLOCK

// ---- Hardware/FBox/FB_Valve.TcPOU
FUNCTION_BLOCK FB_Valve
VAR_INPUT
END_VAR
VAR_OUTPUT
	bDigiOut1 AT %Q* : BOOL;
	bDigiOut2 AT %Q* : BOOL;	//Für Ventile mit 2 Spulen und Mittelstellung
END_VAR
VAR
	
END_VAR

METHOD M_On
VAR_INPUT
	nChannel	: USINT;	//1 oder 2 bei Ventil mit 2 Spulen und Mittelstellung
END_VAR
IF nChannel = 1 THEN
	bDigiOut1 := TRUE;
	bDigiOut2 := FALSE;	
ELSIF nChannel = 2 THEN
	bDigiOut1 := FALSE;
	bDigiOut2 := TRUE;
ELSE
	bDigiOut1 := FALSE;
	bDigiOut2 := FALSE;
END_IF
END_METHOD

METHOD M_Off
VAR_INPUT
END_VAR
bDigiOut1 := FALSE;
bDigiOut2 := FALSE;
END_METHOD

END_FUNCTION_BLOCK

// ---- Hardware/FBox/FB_Pump.TcPOU
FUNCTION_BLOCK FB_Pump
VAR_INPUT
END_VAR
VAR_OUTPUT
END_VAR
VAR
	rStartSpeed		: UINT;		//Startdrehzahl 0..100%
	rRatedSpeed		: UINT;		//Nenndrehzahl 0..100%
	tStartDelay		: TIME;		//Delay Startdrehzahl -> Nenndrehzahl
	timer			: TON;		
	bIsOn			: BOOL;
	//Ausgänge für Geräteverknüpfung
	bDigiOut	 	AT %Q* : BOOL;		//Standardpumpe EIN/AUS
	nPWMValue 		AT %Q* : UINT;	//PWM für Drehzahl
END_VAR

METHOD M_On : BOOL
VAR_INPUT
END_VAR
bDigiOut := TRUE;
IF tStartDelay > T#0S AND NOT bIsOn THEN
	nPWMValue := REAL_TO_UINT(32767.0 / 100 * rStartSpeed);
	timer(IN:=TRUE,PT:= tStartDelay);
	IF timer.Q THEN
		timer(IN:=FALSE);
		nPWMValue := REAL_TO_UINT(32767.0 / 100 * rRatedSpeed);
		M_On := TRUE;	
	END_IF
ELSE
	nPWMValue := REAL_TO_UINT(32767.0 / 100 * rRatedSpeed);
	M_On := TRUE;
	bIsOn := TRUE;
END_IF
END_METHOD

PROPERTY P_bIsOn : BOOL
GET
P_bIsOn := bDigiOut;
END_GET
END_PROPERTY

PROPERTY P_nStartSpeed : USINT
SET
IF P_nStartSpeed <= 100 THEN
	rStartSpeed := P_nStartSpeed; 
ELSE
	rStartSpeed := 100;
END_IF
END_SET
END_PROPERTY

PROPERTY P_nRatedSpeed : USINT
SET
IF P_nRatedSpeed <= 100 THEN
	rRatedSpeed := P_nRatedSpeed; 
ELSE
	rRatedSpeed := 100;
END_IF
END_SET
END_PROPERTY

PROPERTY P_nDelay : UINT
SET
tStartDelay := UINT_TO_TIME(P_nDelay);
END_SET
END_PROPERTY

METHOD M_Off
VAR_INPUT
END_VAR
bDigiOut := FALSE;
nPWMValue := 0;
timer(IN:=FALSE);
bIsOn := FALSE;
END_METHOD

END_FUNCTION_BLOCK

// ---- Hardware/LiquidReserve/FB_GearPump.TcPOU
FUNCTION_BLOCK FB_GearPump

VAR_OUTPUT
	bError : BOOL;
	bBusy : BOOL;
END_VAR
VAR
	bPumpConst 		: BOOL;
	bPumpQuantity 	: BOOL;
	nPumpMicroSteps	: DINT;
	nPumpSpeed		: DINT;
	nPumpSpeedNew	: DINT;
	nStateA_Pump	: USINT;
	nStateA_PumpNext: USINT;
	bStop			: BOOL;
	
	fbTMCM6110		: FB_TMCM6110;
	nPumpNr			: USINT;	//wird in M_init gesetzt und wird automatisch mit jeder neuen Instanzierung inkrementiert
END_VAR

VAR_STAT
	nHighestPumpNr : USINT; //Klassenvariable zum inkrementieren von nPumpNr
END_VAR

VAR CONSTANT
	//Konstanten zur Umrechnung von Flow 10tel µl/s in Speed
	cFactorFlowToSpeed	: REAL := 402653184; //16(2ExpPulsdivisor X 2048 X 32 X 16(MicroStepRes) X 24(FullStep/U)
	cDivisorFlowToSpeed	: REAL := 240000000; //16000(Frequ) X 1.5 µl/U(Fördervolumen Pumpe/U) X 10(10telµl)
	//Konstanten zur Umrechnung von Quantity µl in MircoSteps
	cFactorQuantToMicroSteps	: REAL := 25.6; //384 MircoSteps/U / 15 10telµl/U
END_VAR

IF bPumpConst THEN
	bBusy := TRUE;
	A_PumpConst();
	IF nStateA_Pump >= 80 THEN
		IF nStateA_Pump >= 99 THEN
			bError := TRUE;
		END_IF
		nStateA_Pump := 0;
		bPumpConst := FALSE;
	END_IF
ELSIF bPumpQuantity THEN
	bBusy := TRUE;
	A_PumpQuantity();
	IF nStateA_Pump >= 80 THEN
		IF nStateA_Pump >= 99 THEN
			bError := TRUE;
		END_IF
		nStateA_Pump := 0;
		bPumpQuantity := FALSE;
	END_IF
ELSE
	bBusy := FALSE;
	bStop := FALSE;
END_IF

METHOD M_PumpConst : ERRORID
VAR_INPUT
	nFlow	: DINT;
END_VAR
bPumpConst := TRUE;
nPumpSpeedNew := REAL_TO_DINT(DINT_TO_REAL(nFlow) * cFactorFlowToSpeed / cDivisorFlowToSpeed);
bBusy := TRUE;
bStop := FALSE;
END_METHOD

